  MoveL 1393 to (55.08, -253.68, 406.18) mm, rotated rx -19.35 ry -2.23 rz 0.78 deg; joints [0.707, -147.772, -38.266, -73.505, 93.206, -4.557]
  MoveL 1394 to (54.92, -244.83, 403.1) mm, rotated rx -20.06 ry -2.27 rz 0.83 deg; joints [0.671, -146.589, -40.525, -73.146, 93.202, -4.603]
  MoveL 1395 to (54.92, -237.94, 400.5) mm, rotated rx -20.57 ry -2.12 rz 0.8 deg; joints [0.697, -145.611, -42.376, -72.771, 93.012, -4.583]
  MoveL 1396 to (55.12, -232.38, 398.15) mm, rotated rx -20.87 ry -1.81 rz 0.69 deg; joints [0.778, -144.686, -44.129, -72.215, 92.65, -4.505]
  MoveL 1397 to (55.02, -224.7, 395.11) mm, rotated rx -21.78 ry -1 rz 0.4 deg; joints [1.084, -143.801, -45.655, -72.409, 91.674, -4.211]
  MoveL 1398 to (54.73, -214.72, 391.64) mm, rotated rx -21.72 ry -0.41 rz 0.16 deg; joints [1.286, -141.85, -49.637, -70.273, 91.013, -4.009]
  MoveL 1399 to (54.98, -204.84, 387.37) mm, rotated rx -21.69 ry -0.21 rz 0.08 deg; joints [1.294, -140.064, -53.161, -68.489, 90.801, -4]
  MoveL 1400 to (55.25, -194.58, 383.53) mm, rotated rx -21.83 ry -0.78 rz 0.31 deg; joints [0.986, -138.634, -56.017, -67.249, 91.452, -4.307]
  MoveL 1401 to (55.06, -187.74, 380.29) mm, rotated rx -21.75 ry -1.59 rz 0.63 deg; joints [0.622, -137.594, -58.047, -66.253, 92.371, -4.669]
  MoveL 1402 to (55.53, -182.53, 378.45) mm, rotated rx -21.65 ry -2.04 rz 0.81 deg; joints [0.364, -136.863, -59.574, -65.405, 92.9, -4.926]
  MoveL 1403 to (54.81, -174.44, 375.91) mm, rotated rx -21.54 ry -2.47 rz 0.97 deg; joints [0.18, -135.733, -61.956, -64.088, 93.395, -5.109]
  MoveL 1404 to (54.79, -165.46, 371.7) mm, rotated rx -21.28 ry -2.57 rz 1 deg; joints [0.063, -134.251, -64.859, -62.426, 93.54, -5.222]
  MoveL 1405 to (53.02, -160.4, 369) mm, rotated rx -21.41 ry -2.72 rz 1.07 deg; joints [0.097, -133.514, -66.171, -61.987, 93.684, -5.191]
  MoveL 1406 to (55.23, -155.08, 367) mm, rotated rx -21.73 ry -2.58 rz 1.03 deg; joints [-0.042, -133.026, -67.064, -61.898, 93.535, -5.332]
  MoveL 1407 to (54.71, -145.1, 363.45) mm, rotated rx -21.68 ry -2.38 rz 0.94 deg; joints [0.011, -131.654, -69.821, -60.441, 93.311, -5.278]
  MoveL 1408 to (55.13, -137.69, 360.48) mm, rotated rx -21.26 ry -2.44 rz 0.95 deg; joints [-0.118, -130.495, -72.206, -58.809, 93.424, -5.4]
  MoveL 1409 to (55.28, -132.81, 358.42) mm, rotated rx -20.93 ry -2.36 rz 0.9 deg; joints [-0.148, -129.693, -73.844, -57.645, 93.378, -5.425]
  MoveL 1410 to (55.22, -124.84, 355.82) mm, rotated rx -20.86 ry -2.05 rz 0.78 deg; joints [-0.064, -128.673, -75.93, -56.476, 93.029, -5.339]
  MoveL 1411 to (54.98, -114.49, 352.02) mm, rotated rx -20.31 ry -1.65 rz 0.61 deg; joints [0.034, -127.128, -79.135, -54.23, 92.636, -5.231]
  MoveL 1412 to (59.43, -108.23, 350) mm, rotated rx -20.42 ry -1.45 rz 0.54 deg; joints [-0.284, -126.59, -80.24, -53.769, 92.469, -5.547]
  MoveL 1413 to (54.78, -104.7, 347.81) mm, rotated rx -20.44 ry -1.33 rz 0.49 deg; joints [0.126, -125.933, -81.347, -53.307, 92.267, -5.142]
  MoveL 1414 to (54.83, -96.04, 345.13) mm, rotated rx -20.42 ry -1.17 rz 0.44 deg; joints [0.128, -124.985, -83.305, -52.268, 92.1, -5.139]
  MoveL 1415 to (55.03, -86.29, 340.97) mm, rotated rx -20.38 ry -1.02 rz 0.38 deg; joints [0.101, -123.809, -85.531, -51.167, 91.946, -5.164]
  MoveL 1416 to (55.31, -80.99, 339) mm, rotated rx -20.5 ry -1.09 rz 0.41 deg; joints [0.003, -123.296, -86.506, -50.831, 92.03, -5.263]
  MoveL 1417 to (54.95, -74.37, 337.02) mm, rotated rx -20.6 ry -1.3 rz 0.49 deg; joints [-0.12, -122.697, -87.74, -50.318, 92.266, -5.387]
  MoveL 1418 to (55.01, -64.82, 333.24) mm, rotated rx -20.62 ry -1.46 rz 0.55 deg; joints [-0.287, -121.687, -89.671, -49.444, 92.457, -5.553]
  MoveL 1419 to (54.85, -58, 330.46) mm, rotated rx -20.53 ry -1.63 rz 0.61 deg; joints [-0.429, -120.927, -91.145, -48.659, 92.676, -5.693]
  MoveL 1420 to (55.08, -53.48, 328.66) mm, rotated rx -20.28 ry -1.75 rz 0.65 deg; joints [-0.563, -120.374, -92.289, -47.834, 92.845, -5.822]
  MoveL 1421 to (54.97, -45.34, 325.78) mm, rotated rx -19.8 ry -1.75 rz 0.63 deg; joints [-0.651, -119.376, -94.415, -46.232, 92.899, -5.9]
  MoveL 1422 to (55, -34.77, 321.83) mm, rotated rx -19.25 ry -1.73 rz 0.6 deg; joints [-0.776, -118.117, -97.048, -44.316, 92.948, -6.012]
  MoveL 1423 to (55.17, -28.7, 320) mm, rotated rx -19.04 ry -1.82 rz 0.63 deg; joints [-0.917, -117.517, -98.38, -43.388, 93.099, -6.147]
  MoveL 1424 to (54.83, -23.54, 318) mm, rotated rx -19.21 ry -1.88 rz 0.65 deg; joints [-0.959, -117.05, -99.206, -43.208, 93.144, -6.193]
  MoveL 1425 to (55.14, -14.22, 315.38) mm, rotated rx -19.3 ry -1.62 rz 0.57 deg; joints [-0.947, -116.239, -100.898, -42.396, 92.866, -6.182]
  MoveL 1426 to (54.99, -4.33, 311.44) mm, rotated rx -19.09 ry -1.52 rz 0.53 deg; joints [-1, -115.16, -103.001, -41.15, 92.788, -6.229]
  MoveL 1427 to (55.02, 5.42, 307.78) mm, rotated rx -18.68 ry -1.44 rz 0.49 deg; joints [-1.098, -114.093, -105.207, -39.596, 92.77, -6.316]
  MoveL 1428 to (55.05, 14.94, 305) mm, rotated rx -18.73 ry -1.36 rz 0.46 deg; joints [-1.159, -113.294, -106.879, -38.769, 92.685, -6.377]
  MoveL 1429 to (54.97, 24.93, 302.19) mm, rotated rx -18.4 ry -1.17 rz 0.39 deg; joints [-1.181, -112.36, -108.994, -37.237, 92.527, -6.39]
  MoveL 1430 to (55.25, 31.9, 300) mm, rotated rx -18.6 ry -1.02 rz 0.34 deg; joints [-1.192, -111.805, -110.057, -36.92, 92.345, -6.405]
  MoveL 1431 to (54.96, 36.41, 298.4) mm, rotated rx -18.88 ry -0.94 rz 0.32 deg; joints [-1.157, -111.448, -110.635, -36.964, 92.23, -6.376]
  MoveL 1432 to (54.92, 44.41, 294.89) mm, rotated rx -18.74 ry -0.71 rz 0.24 deg; joints [-1.131, -110.564, -112.252, -36.062, 92.003, -6.347]
  MoveL 1433 to (55.12, 54.76, 291.8) mm, rotated rx -18.4 ry -0.72 rz 0.24 deg; joints [-1.309, -109.656, -114.303, -34.594, 92.079, -6.513]
  MoveL 1434 to (55.11, 61.12, 290) mm, rotated rx -17.74 ry -0.7 rz 0.22 deg; joints [-1.422, -109.017, -115.958, -32.921, 92.152, -6.608]
  MoveL 1435 to (54.8, 66.06, 288.46) mm, rotated rx -17.44 ry -0.7 rz 0.22 deg; joints [-1.477, -108.55, -117.066, -31.98, 92.204, -6.655]
  MoveL 1436 to (54.9, 74.97, 284.68) mm, rotated rx -17.22 ry -0.7 rz 0.22 deg; joints [-1.639, -107.658, -118.76, -30.971, 92.264, -6.807]
  MoveL 1437 to (55.21, 85.34, 282.5) mm, rotated rx -17.34 ry -0.69 rz 0.21 deg; joints [-1.8, -107.029, -120.321, -30.158, 92.267, -6.968]
  MoveL 1438 to (54.78, 93.08, 280.4) mm, rotated rx -17.02 ry -0.27 rz 0.08 deg; joints [-1.61, -106.334, -121.989, -28.813, 91.826, -6.771]
  MoveL 1439 to (57.07, 97.19, 278.81) mm, rotated rx -16.4 ry 0.04 rz -0.01 deg; joints [-1.792, -105.907, -123.158, -27.418, 91.62, -6.931]
  MoveL 1440 to (58.78, 100.67, 277.75) mm, rotated rx -16.4 ry 0.12 rz -0.04 deg; joints [-2.002, -105.698, -123.644, -27.142, 91.586, -7.135]
  MoveL 1441 to (64.56, -260.81, 408.44) mm, rotated rx -18.59 ry -2.72 rz 0.92 deg; joints [-0.095, -149.152, -35.66, -74.064, 93.927, -5.336]
  MoveL 1442 to (65.01, -254.78, 407.2) mm, rotated rx -18.39 ry -2.66 rz 0.88 deg; joints [-0.144, -147.728, -38.763, -72.186, 93.883, -5.38]
  MoveL 1443 to (64.96, -244.73, 403.18) mm, rotated rx -20.08 ry -2.38 rz 0.87 deg; joints [-0.057, -147.081, -39.585, -73.668, 93.443, -5.322]
  MoveL 1444 to (65.61, -236.7, 401.03) mm, rotated rx -21.08 ry -2.09 rz 0.8 deg; joints [-0.012, -146.4, -40.839, -74.057, 93.047, -5.29]
  MoveL 1445 to (62.2, -232.13, 398.8) mm, rotated rx -21.47 ry -1.65 rz 0.65 deg; joints [0.37, -145.511, -42.445, -73.672, 92.498, -4.916]
  MoveL 1446 to (64.8, -224.8, 395.47) mm, rotated rx -22.46 ry -1.21 rz 0.5 deg; joints [0.345, -144.896, -43.381, -74.313, 91.947, -4.951]
  MoveL 1447 to (65.02, -216.02, 391.48) mm, rotated rx -22.19 ry -1.01 rz 0.41 deg; joints [0.343, -142.892, -47.393, -72.019, 91.755, -4.949]
  MoveL 1448 to (67.07, -211.79, 389) mm, rotated rx -22.21 ry -1.04 rz 0.42 deg; joints [0.156, -142.13, -48.809, -71.388, 91.813, -5.134]
  MoveL 1449 to (64.92, -205.17, 386.05) mm, rotated rx -21.61 ry -0.79 rz 0.31 deg; joints [0.347, -140.361, -52.43, -68.915, 91.563, -4.938]
  MoveL 1450 to (64.99, -195.38, 382.72) mm, rotated rx -20.75 ry -1.55 rz 0.59 deg; joints [-0.061, -138.394, -56.676, -65.857, 92.509, -5.332]
  MoveL 1451 to (64.36, -188.78, 380.15) mm, rotated rx -20.94 ry -2.09 rz 0.8 deg; joints [-0.279, -137.586, -58.253, -65.334, 93.099, -5.553]
  MoveL 1452 to (65.35, -183.29, 378.42) mm, rotated rx -21.31 ry -2.24 rz 0.87 deg; joints [-0.445, -137.108, -59.179, -65.283, 93.259, -5.723]
  MoveL 1453 to (65.07, -174.7, 376.9) mm, rotated rx -21.54 ry -2.09 rz 0.83 deg; joints [-0.417, -136.146, -61.303, -64.327, 93.079, -5.698]
  MoveL 1454 to (65.38, -165.59, 372.14) mm, rotated rx -21.23 ry -1.93 rz 0.75 deg; joints [-0.455, -134.518, -64.428, -62.516, 92.93, -5.731]
  MoveL 1455 to (65.07, -160.4, 369) mm, rotated rx -21.45 ry -1.96 rz 0.77 deg; joints [-0.488, -133.793, -65.634, -62.25, 92.959, -5.766]
  MoveL 1456 to (64.92, -155.17, 367.35) mm, rotated rx -21.91 ry -1.93 rz 0.78 deg; joints [-0.486, -133.373, -66.4, -62.362, 92.88, -5.771]
  MoveL 1457 to (65.21, -145.15, 364.29) mm, rotated rx -21.56 ry -2.01 rz 0.79 deg; joints [-0.634, -131.962, -69.413, -60.425, 93.014, -5.914]
  MoveL 1458 to (65.04, -137.22, 360.8) mm, rotated rx -21.12 ry -2.22 rz 0.86 deg; joints [-0.801, -130.701, -71.962, -58.731, 93.304, -6.073]
  MoveL 1459 to (64.64, -132.44, 358.36) mm, rotated rx -21.09 ry -2.27 rz 0.88 deg; joints [-0.84, -130.015, -73.227, -58.128, 93.37, -6.112]
  MoveL 1460 to (65.05, -125.09, 356.02) mm, rotated rx -21.31 ry -2.11 rz 0.82 deg; joints [-0.856, -129.253, -74.741, -57.58, 93.181, -6.13]
  MoveL 1461 to (65.01, -114.69, 352.96) mm, rotated rx -20.63 ry -1.66 rz 0.62 deg; joints [-0.764, -127.702, -78.121, -55.022, 92.744, -6.025]
  MoveL 1462 to (65.64, -107.48, 350.37) mm, rotated rx -20.58 ry -1.42 rz 0.53 deg; joints [-0.776, -126.837, -79.857, -54.086, 92.504, -6.036]
  MoveL 1463 to (65.06, -102.58, 347.84) mm, rotated rx -20.65 ry -1.33 rz 0.5 deg; joints [-0.732, -126.192, -80.984, -53.659, 92.393, -5.992]
  MoveL 1464 to (64.8, -95.29, 344.81) mm, rotated rx -20.52 ry -1.19 rz 0.45 deg; joints [-0.719, -125.245, -82.829, -52.616, 92.255, -5.977]
  MoveL 1465 to (65.28, -85.57, 341) mm, rotated rx -20.49 ry -0.96 rz 0.36 deg; joints [-0.744, -124.11, -85.034, -51.495, 92.02, -6]
  MoveL 1466 to (64.1, -80.02, 339) mm, rotated rx -20.41 ry -0.96 rz 0.36 deg; joints [-0.699, -123.442, -86.371, -50.745, 92.019, -5.955]
  MoveL 1467 to (64.98, -74.27, 337.4) mm, rotated rx -20.3 ry -0.9 rz 0.33 deg; joints [-0.802, -122.854, -87.664, -49.919, 91.98, -6.053]
  MoveL 1468 to (65.02, -64.62, 333.14) mm, rotated rx -20.29 ry -1.17 rz 0.43 deg; joints [-1.039, -121.794, -89.629, -49.048, 92.308, -6.289]
  MoveL 1469 to (65.63, -57.19, 330.53) mm, rotated rx -20.07 ry -1.48 rz 0.54 deg; joints [-1.332, -121.022, -91.254, -48.024, 92.701, -6.575]
  MoveL 1470 to (64.51, -52.14, 329) mm, rotated rx -20.17 ry -1.71 rz 0.63 deg; joints [-1.398, -120.58, -92.152, -47.693, 92.95, -6.644]
  MoveL 1471 to (64.89, -44.96, 327.12) mm, rotated rx -19.87 ry -1.72 rz 0.62 deg; joints [-1.528, -119.845, -93.836, -46.456, 93.013, -6.766]
  MoveL 1472 to (64.91, -34.85, 322.66) mm, rotated rx -19.27 ry -1.62 rz 0.57 deg; joints [-1.632, -118.522, -96.488, -44.523, 92.99, -6.855]
  MoveL 1473 to (65.83, -28.11, 320) mm, rotated rx -19.11 ry -1.5 rz 0.52 deg; joints [-1.744, -117.792, -97.937, -43.641, 92.9, -6.961]
  MoveL 1474 to (64.59, -23.19, 318.3) mm, rotated rx -19.34 ry -1.45 rz 0.51 deg; joints [-1.652, -117.347, -98.733, -43.502, 92.812, -6.875]
  MoveL 1475 to (65.09, -14.35, 315.73) mm, rotated rx -19.48 ry -1.32 rz 0.47 deg; joints [-1.724, -116.61, -100.249, -42.856, 92.668, -6.949]
  MoveL 1476 to (65, -4.36, 312.96) mm, rotated rx -19.17 ry -1.29 rz 0.45 deg; joints [-1.838, -115.661, -102.395, -41.349, 92.691, -7.053]
  MoveL 1477 to (67.12, 1.57, 310) mm, rotated rx -18.88 ry -1.26 rz 0.43 deg; joints [-2.128, -114.98, -103.691, -40.453, 92.745, -7.332]
  MoveL 1478 to (64.74, 5.9, 307.87) mm, rotated rx -18.76 ry -1.19 rz 0.4 deg; joints [-1.922, -114.379, -104.765, -39.846, 92.647, -7.127]
  MoveL 1479 to (64.99, 14.9, 305.22) mm, rotated rx -18.7 ry -1.07 rz 0.36 deg; joints [-2.006, -113.595, -106.445, -38.879, 92.553, -7.206]
  MoveL 1480 to (64.96, 25.12, 302.15) mm, rotated rx -18.59 ry -1.1 rz 0.37 deg; joints [-2.163, -112.716, -108.34, -37.765, 92.624, -7.358]
  MoveL 1481 to (64.3, 31.36, 300) mm, rotated rx -18.81 ry -1.09 rz 0.37 deg; joints [-2.163, -112.197, -109.276, -37.566, 92.587, -7.363]
  MoveL 1482 to (65.2, 36.26, 297.42) mm, rotated rx -19.08 ry -1.06 rz 0.37 deg; joints [-2.298, -111.741, -109.881, -37.689, 92.549, -7.502]
  MoveL 1483 to (65.02, 45.12, 295.08) mm, rotated rx -18.74 ry -1.03 rz 0.35 deg; joints [-2.407, -110.963, -111.72, -36.29, 92.574, -7.602]
  MoveL 1484 to (64.94, 54.73, 292.15) mm, rotated rx -18.47 ry -1.1 rz 0.37 deg; joints [-2.61, -110.134, -113.576, -35.015, 92.73, -7.795]
  MoveL 1485 to (63.94, 60.82, 290) mm, rotated rx -17.96 ry -1.03 rz 0.33 deg; joints [-2.59, -109.442, -115.145, -33.614, 92.712, -7.76]
  MoveL 1486 to (65.16, 65.51, 288.44) mm, rotated rx -17.52 ry -0.96 rz 0.3 deg; joints [-2.795, -108.996, -116.265, -32.505, 92.744, -7.948]
  MoveL 1487 to (64.96, 75.06, 285.39) mm, rotated rx -17.35 ry -0.63 rz 0.2 deg; joints [-2.738, -108.132, -118.107, -31.313, 92.412, -7.884]
  MoveL 1488 to (65.01, 85.34, 282.44) mm, rotated rx -17.3 ry -0.39 rz 0.12 deg; joints [-2.761, -107.319, -119.899, -30.253, 92.171, -7.904]
  MoveL 1489 to (64.71, 92.06, 280.15) mm, rotated rx -17.29 ry -0.5 rz 0.16 deg; joints [-2.917, -106.779, -120.993, -29.708, 92.321, -8.057]
  MoveL 1490 to (65.23, 97.05, 278.32) mm, rotated rx -16.92 ry -0.44 rz 0.13 deg; joints [-3.067, -106.307, -122.11, -28.689, 92.347, -8.191]
  MoveL 1491 to (65.21, 101.45, 276.39) mm, rotated rx -16.78 ry -0.11 rz 0.03 deg; joints [-2.937, -105.802, -123.062, -28.05, 91.99, -8.058]
  MoveL 1492 to (75.11, -263.32, 410.7) mm, rotated rx -19.34 ry -1.95 rz 0.68 deg; joints [-0.467, -151.14, -31.599, -76.835, 93.119, -5.711]
  MoveL 1493 to (80.87, -259.66, 410) mm, rotated rx -18.89 ry -2.65 rz 0.91 deg; joints [-1.154, -150.329, -33.526, -75.386, 94.028, -6.384]
  MoveL 1494 to (75.51, -259.66, 410) mm, rotated rx -18.52 ry -2.32 rz 0.78 deg; joints [-0.683, -149.52, -35.241, -74.043, 93.622, -5.91]
  MoveL 1495 to (75.18, -253.52, 407.14) mm, rotated rx -18.5 ry -2.65 rz 0.89 deg; joints [-0.833, -148.106, -38.068, -72.657, 93.999, -6.06]
  MoveL 1496 to (74.85, -244.56, 402.65) mm, rotated rx -20.82 ry -2.61 rz 0.99 deg; joints [-0.798, -148.266, -36.982, -75.881, 93.751, -6.068]
  MoveL 1497 to (75.1, -236.23, 401.3) mm, rotated rx -21.65 ry -2.25 rz 0.89 deg; joints [-0.706, -147.409, -38.764, -75.751, 93.279, -5.988]
  MoveL 1498 to (75.24, -225.13, 395.22) mm, rotated rx -22.62 ry -2.19 rz 0.91 deg; joints [-0.755, -145.769, -41.608, -75.508, 93.139, -6.049]
  MoveL 1499 to (75.24, -216.09, 391.13) mm, rotated rx -22.66 ry -1.94 rz 0.81 deg; joints [-0.725, -143.894, -45.288, -73.718, 92.856, -6.018]
  MoveL 1500 to (73.17, -211.79, 389) mm, rotated rx -22.42 ry -1.54 rz 0.64 deg; joints [-0.465, -142.659, -47.738, -72.212, 92.417, -5.755]
  MoveL 1501 to (75.03, -204.96, 386.98) mm, rotated rx -21.4 ry -1.74 rz 0.68 deg; joints [-0.76, -140.874, -51.676, -69.076, 92.76, -6.034]
  MoveL 1502 to (75.1, -194.69, 383.85) mm, rotated rx -20.24 ry -1.83 rz 0.67 deg; joints [-0.922, -138.535, -56.799, -65.146, 92.989, -6.176]
  MoveL 1503 to (75.37, -187.45, 380.54) mm, rotated rx -20.91 ry -1.7 rz 0.65 deg; joints [-0.928, -137.788, -58.037, -65.311, 92.79, -6.192]
  MoveL 1504 to (74.68, -182.22, 378.28) mm, rotated rx -21.5 ry -1.62 rz 0.64 deg; joints [-0.87, -137.312, -58.79, -65.613, 92.643, -6.144]
  MoveL 1505 to (74.95, -174.56, 376.81) mm, rotated rx -21.88 ry -1.3 rz 0.52 deg; joints [-0.797, -136.526, -60.478, -65.05, 92.246, -6.076]
  MoveL 1506 to (75.03, -164.4, 371.69) mm, rotated rx -21.14 ry -0.97 rz 0.37 deg; joints [-0.783, -134.451, -64.613, -62.222, 91.966, -6.049]
  MoveL 1507 to (75.88, -158.9, 370) mm, rotated rx -21.36 ry -0.93 rz 0.36 deg; joints [-0.869, -133.892, -65.735, -61.876, 91.919, -6.138]
  MoveL 1508 to (74.82, -154.25, 367.84) mm, rotated rx -21.66 ry -1.25 rz 0.5 deg; joints [-0.956, -133.412, -66.553, -61.873, 92.243, -6.23]
  MoveL 1509 to (75.16, -145.64, 365.57) mm, rotated rx -21.37 ry -1.63 rz 0.64 deg; joints [-1.23, -132.313, -68.983, -60.309, 92.714, -6.499]
  MoveL 1510 to (75.18, -136.04, 361.41) mm, rotated rx -21.02 ry -1.56 rz 0.6 deg; joints [-1.311, -130.841, -71.918, -58.497, 92.692, -6.572]
  MoveL 1511 to (74.07, -131.61, 358.88) mm, rotated rx -21.06 ry -1.58 rz 0.61 deg; joints [-1.277, -130.175, -73.085, -58.029, 92.702, -6.54]
  MoveL 1512 to (74.88, -125, 356.05) mm, rotated rx -21.49 ry -1.58 rz 0.62 deg; joints [-1.388, -129.57, -74.116, -58.043, 92.675, -6.657]
  MoveL 1513 to (75.04, -114.51, 352.44) mm, rotated rx -21.12 ry -1.33 rz 0.51 deg; joints [-1.405, -128.125, -77.123, -56.081, 92.447, -6.666]
  MoveL 1514 to (74.03, -107.97, 350.43) mm, rotated rx -20.83 ry -1.07 rz 0.41 deg; joints [-1.282, -127.196, -79.103, -54.703, 92.187, -6.538]
  MoveL 1515 to (75.51, -103.23, 347.77) mm, rotated rx -20.74 ry -0.91 rz 0.35 deg; joints [-1.385, -126.535, -80.291, -54.079, 92.043, -6.638]
  MoveL 1516 to (75, -94.89, 345.05) mm, rotated rx -20.65 ry -0.85 rz 0.32 deg; joints [-1.402, -125.565, -82.294, -52.943, 91.988, -6.652]
  MoveL 1517 to (74.92, -84.51, 341.34) mm, rotated rx -20.72 ry -0.72 rz 0.27 deg; joints [-1.437, -124.438, -84.516, -51.909, 91.848, -6.688]
  MoveL 1518 to (75.1, -74.48, 337.81) mm, rotated rx -20.46 ry -0.55 rz 0.21 deg; joints [-1.49, -123.242, -86.983, -50.358, 91.706, -6.735]
  MoveL 1519 to (75, -64.84, 333.79) mm, rotated rx -19.97 ry -0.47 rz 0.17 deg; joints [-1.578, -121.963, -89.57, -48.554, 91.696, -6.811]
  MoveL 1520 to (75.02, -56.43, 330.96) mm, rotated rx -19.78 ry -0.67 rz 0.24 deg; joints [-1.78, -121.084, -91.416, -47.426, 91.958, -7.007]
  MoveL 1521 to (74.42, -51.73, 329) mm, rotated rx -19.89 ry -0.86 rz 0.31 deg; joints [-1.874, -120.632, -92.222, -47.219, 92.165, -7.103]
  MoveL 1522 to (75.01, -45.45, 326.52) mm, rotated rx -19.84 ry -0.94 rz 0.34 deg; joints [-2.045, -119.987, -93.482, -46.568, 92.283, -7.27]
  MoveL 1523 to (75.01, -34.99, 324.07) mm, rotated rx -19.45 ry -0.83 rz 0.29 deg; joints [-2.135, -118.954, -95.906, -44.775, 92.234, -7.35]
  MoveL 1524 to (74.93, -27.07, 320.43) mm, rotated rx -19.19 ry -0.7 rz 0.24 deg; joints [-2.178, -117.977, -97.768, -43.622, 92.129, -7.385]
  MoveL 1525 to (74.92, -21.92, 318.61) mm, rotated rx -19.29 ry -0.81 rz 0.28 deg; joints [-2.299, -117.533, -98.621, -43.325, 92.261, -7.507]
  MoveL 1526 to (75.04, -14.29, 315.6) mm, rotated rx -19.5 ry -0.98 rz 0.35 deg; joints [-2.488, -116.867, -99.812, -43.038, 92.444, -7.7]
  MoveL 1527 to (74.96, -4.46, 312.76) mm, rotated rx -19.02 ry -1.05 rz 0.36 deg; joints [-2.685, -115.891, -102.049, -41.327, 92.621, -7.882]
  MoveL 1528 to (75.69, 3.3, 310) mm, rotated rx -19.07 ry -0.99 rz 0.34 deg; joints [-2.829, -115.198, -103.408, -40.705, 92.572, -8.024]
  MoveL 1529 to (74.23, 7.81, 308.64) mm, rotated rx -18.97 ry -0.95 rz 0.33 deg; joints [-2.736, -114.727, -104.41, -40.063, 92.529, -7.93]
  MoveL 1530 to (74.94, 14.96, 305.92) mm, rotated rx -18.83 ry -0.86 rz 0.29 deg; joints [-2.875, -114.021, -105.828, -39.204, 92.482, -8.062]
  MoveL 1531 to (74.99, 25.08, 302.55) mm, rotated rx -18.4 ry -0.92 rz 0.31 deg; joints [-3.101, -113.04, -107.984, -37.628, 92.647, -8.273]
  MoveL 1532 to (76.15, 31.98, 300.05) mm, rotated rx -18.82 ry -1.04 rz 0.36 deg; joints [-3.368, -112.587, -108.722, -37.782, 92.764, -8.547]
  MoveL 1533 to (74.3, 36.05, 298.14) mm, rotated rx -19.01 ry -1.09 rz 0.37 deg; joints [-3.257, -112.153, -109.372, -37.758, 92.761, -8.444]
  MoveL 1534 to (75.11, 44.67, 295.69) mm, rotated rx -18.62 ry -1.21 rz 0.41 deg; joints [-3.586, -111.431, -111.107, -36.397, 93.009, -8.758]
  MoveL 1535 to (74.88, 54.68, 291.77) mm, rotated rx -18.37 ry -1.5 rz 0.5 deg; joints [-3.935, -110.497, -112.979, -35.272, 93.415, -9.096]
  MoveL 1536 to (74.13, 60.4, 290) mm, rotated rx -18.17 ry -1.49 rz 0.49 deg; joints [-3.97, -109.967, -114.156, -34.433, 93.443, -9.124]
  MoveL 1537 to (75.11, 64.93, 288.79) mm, rotated rx -18.05 ry -1.28 rz 0.42 deg; joints [-4.04, -109.604, -115.028, -33.769, 93.255, -9.186]
  MoveL 1538 to (74.84, 75.3, 285.59) mm, rotated rx -17.67 ry -0.8 rz 0.25 deg; joints [-3.939, -108.617, -117.239, -32.091, 92.792, -9.071]
  MoveL 1539 to (75.02, 85.38, 282.27) mm, rotated rx -17.28 ry -0.74 rz 0.23 deg; joints [-4.16, -107.739, -119.233, -30.587, 92.845, -9.273]
  MoveL 1540 to (75.39, 92.51, 280.32) mm, rotated rx -17.48 ry -0.57 rz 0.18 deg; joints [-4.21, -107.252, -120.243, -30.241, 92.644, -9.328]
  MoveL 1541 to (73.93, 97.03, 278.51) mm, rotated rx -17.35 ry -0.42 rz 0.13 deg; joints [-4.047, -106.74, -121.234, -29.597, 92.474, -9.162]
  MoveL 1542 to (73.9, 100.81, 277.62) mm, rotated rx -17.26 ry -0.3 rz 0.09 deg; joints [-4.05, -106.463, -121.947, -29.052, 92.369, -9.161]
  MoveL 1543 to (84.62, -262.23, 410) mm, rotated rx -19.74 ry -3.1 rz 1.11 deg; joints [-1.525, -152.298, -29.177, -78.689, 94.488, -6.771]
  MoveL 1544 to (85.18, -254.45, 406.95) mm, rotated rx -19.33 ry -3.17 rz 1.11 deg; joints [-1.669, -149.81, -34.361, -75.601, 94.625, -6.905]
  MoveL 1545 to (84.93, -244.07, 403.5) mm, rotated rx -21.32 ry -2.99 rz 1.16 deg; joints [-1.6, -149.493, -34.573, -77.657, 94.224, -6.875]
  MoveL 1546 to (84.92, -235.7, 402.03) mm, rotated rx -22.08 ry -2.73 rz 1.11 deg; joints [-1.539, -148.503, -36.641, -77.308, 93.863, -6.824]
  MoveL 1547 to (84.8, -224.66, 395.97) mm, rotated rx -22.6 ry -2.59 rz 1.08 deg; joints [-1.562, -146.344, -40.642, -75.969, 93.667, -6.854]
  MoveL 1548 to (85.07, -214.39, 391.74) mm, rotated rx -22.83 ry -2.65 rz 1.12 deg; joints [-1.688, -144.494, -44.298, -74.403, 93.726, -6.983]
  MoveL 1549 to (86.97, -207.97, 390) mm, rotated rx -21.77 ry -3 rz 1.2 deg; joints [-2.055, -142.69, -48.316, -71.198, 94.257, -7.334]
  MoveL 1550 to (90.52, -207.58, 390) mm, rotated rx -21.73 ry -3.09 rz 1.23 deg; joints [-2.341, -142.798, -48.151, -71.253, 94.395, -7.619]
  MoveL 1551 to (84.6, -203.52, 388.23) mm, rotated rx -21.16 ry -2.83 rz 1.1 deg; joints [-1.888, -141.306, -51.227, -69.033, 94.118, -7.156]
  MoveL 1552 to (85.05, -194.33, 384.67) mm, rotated rx -20.74 ry -2.35 rz 0.89 deg; joints [-1.83, -139.426, -55.091, -66.575, 93.638, -7.086]
  MoveL 1553 to (85.62, -185.53, 380.69) mm, rotated rx -21.69 ry -1.5 rz 0.6 deg; joints [-1.569, -138.461, -56.672, -66.792, 92.592, -6.84]
  MoveL 1554 to (83.88, -181.16, 378.92) mm, rotated rx -22.09 ry -1.17 rz 0.48 deg; joints [-1.332, -137.911, -57.642, -66.725, 92.163, -6.609]
  MoveL 1555 to (85.03, -174.6, 376.81) mm, rotated rx -22.34 ry -0.68 rz 0.28 deg; joints [-1.258, -137.07, -59.321, -66.066, 91.599, -6.537]
  MoveL 1556 to (85.14, -164.6, 371.9) mm, rotated rx -21.31 ry -0.54 rz 0.21 deg; joints [-1.346, -134.868, -63.812, -62.74, 91.573, -6.607]
  MoveL 1557 to (85.07, -158.9, 370) mm, rotated rx -21.03 ry -0.63 rz 0.24 deg; joints [-1.446, -133.974, -65.713, -61.469, 91.721, -6.701]
  MoveL 1558 to (85.04, -154.1, 367.79) mm, rotated rx -20.99 ry -0.8 rz 0.31 deg; joints [-1.563, -133.299, -67.009, -60.834, 91.917, -6.817]
  MoveL 1559 to (85.13, -145.29, 365.23) mm, rotated rx -21.13 ry -1.21 rz 0.47 deg; joints [-1.827, -132.389, -68.917, -60.035, 92.387, -7.083]
  MoveL 1560 to (84.92, -135.28, 361.14) mm, rotated rx -21.24 ry -1.25 rz 0.48 deg; joints [-1.923, -131.137, -71.329, -58.997, 92.422, -7.181]
  MoveL 1561 to (84.88, -124.93, 356.15) mm, rotated rx -21.55 ry -1 rz 0.4 deg; joints [-1.912, -129.839, -73.641, -58.257, 92.126, -7.174]
  MoveL 1562 to (85, -114.4, 352.4) mm, rotated rx -21.39 ry -0.85 rz 0.33 deg; joints [-1.971, -128.491, -76.384, -56.687, 91.991, -7.229]
  MoveL 1563 to (85.47, -107.67, 350.29) mm, rotated rx -21.16 ry -0.75 rz 0.29 deg; joints [-2.047, -127.64, -78.203, -55.483, 91.924, -7.299]
  MoveL 1564 to (84.68, -102.56, 348.03) mm, rotated rx -21.01 ry -0.59 rz 0.23 deg; joints [-1.973, -126.884, -79.671, -54.597, 91.757, -7.223]
  MoveL 1565 to (84.73, -94.7, 345.08) mm, rotated rx -20.69 ry -0.4 rz 0.15 deg; joints [-1.994, -125.818, -81.869, -53.117, 91.598, -7.236]
  MoveL 1566 to (85.2, -84.82, 341.13) mm, rotated rx -20.7 ry -0.44 rz 0.17 deg; joints [-2.164, -124.718, -83.994, -52.114, 91.664, -7.404]
  MoveL 1567 to (85.17, -74.33, 337.43) mm, rotated rx -20.66 ry -0.5 rz 0.19 deg; joints [-2.315, -123.596, -86.253, -50.952, 91.758, -7.553]
  MoveL 1568 to (84.97, -64.89, 333.9) mm, rotated rx -20.2 ry -0.07 rz 0.03 deg; joints [-2.233, -122.329, -88.878, -49.076, 91.354, -7.46]
  MoveL 1569 to (84.98, -56.59, 331.06) mm, rotated rx -19.62 ry 0.22 rz -0.08 deg; joints [-2.226, -121.234, -91.26, -47.177, 91.122, -7.44]
  MoveL 1570 to (85.06, -51.84, 328.83) mm, rotated rx -19.58 ry 0.11 rz -0.04 deg; joints [-2.351, -120.695, -92.251, -46.695, 91.262, -7.561]
  MoveL 1571 to (85.07, -45.47, 326.64) mm, rotated rx -19.64 ry -0.11 rz 0.04 deg; joints [-2.538, -120.128, -93.373, -46.24, 91.516, -7.748]
  MoveL 1572 to (85.07, -35, 324) mm, rotated rx -19.61 ry -0.34 rz 0.12 deg; joints [-2.79, -119.257, -95.33, -45.167, 91.809, -7.997]
  MoveL 1573 to (84.43, -27.54, 320.55) mm, rotated rx -19.07 ry -0.49 rz 0.17 deg; joints [-2.954, -118.266, -97.328, -43.649, 92.071, -8.144]
  MoveL 1574 to (85.15, -22.51, 318.39) mm, rotated rx -19.02 ry -0.56 rz 0.19 deg; joints [-3.138, -117.763, -98.28, -43.174, 92.191, -8.325]
  MoveL 1575 to (85.09, -14.25, 315.9) mm, rotated rx -19.33 ry -0.59 rz 0.21 deg; joints [-3.244, -117.132, -99.515, -42.88, 92.198, -8.437]
  MoveL 1576 to (84.98, -4.26, 312.2) mm, rotated rx -18.98 ry -0.91 rz 0.31 deg; joints [-3.583, -116.127, -101.611, -41.509, 92.644, -8.763]
  MoveL 1577 to (82.62, 2.29, 310) mm, rotated rx -19.05 ry -1.02 rz 0.35 deg; joints [-3.512, -115.492, -102.844, -40.993, 92.738, -8.696]
  MoveL 1578 to (85.48, 6.19, 308.36) mm, rotated rx -19.06 ry -1.13 rz 0.39 deg; joints [-3.912, -115.227, -103.352, -40.796, 92.92, -9.091]
  MoveL 1579 to (84.99, 14.95, 306.4) mm, rotated rx -18.9 ry -1.12 rz 0.38 deg; joints [-4.009, -114.512, -105.069, -39.637, 92.952, -9.182]
  MoveL 1580 to (84.93, 24.98, 302.2) mm, rotated rx -18.3 ry -1.09 rz 0.36 deg; joints [-4.217, -113.368, -107.434, -37.833, 93.055, -9.367]
  MoveL 1581 to (84.61, 32.85, 300.05) mm, rotated rx -18.72 ry -1.15 rz 0.39 deg; joints [-4.316, -112.86, -108.411, -37.792, 93.066, -9.478]
  MoveL 1582 to (85.33, 37.25, 298.87) mm, rotated rx -18.93 ry -1.25 rz 0.43 deg; joints [-4.512, -112.623, -108.9, -37.773, 93.184, -9.678]
  MoveL 1583 to (85.08, 44.63, 296.09) mm, rotated rx -18.5 ry -1.28 rz 0.43 deg; joints [-4.681, -111.847, -110.573, -36.465, 93.312, -9.831]
  MoveL 1584 to (85.01, 54.71, 292.37) mm, rotated rx -18.28 ry -1.28 rz 0.42 deg; joints [-4.894, -110.904, -112.497, -35.28, 93.39, -10.032]
  MoveL 1585 to (85.16, 61.25, 290.32) mm, rotated rx -18.54 ry -1.06 rz 0.36 deg; joints [-4.885, -110.403, -113.436, -35.055, 93.12, -10.03]
  MoveL 1586 to (84.98, 66.19, 288.57) mm, rotated rx -18.39 ry -0.9 rz 0.3 deg; joints [-4.88, -109.912, -114.461, -34.349, 92.971, -10.019]
  MoveL 1587 to (84.99, 75.45, 285.6) mm, rotated rx -17.77 ry -0.97 rz 0.31 deg; joints [-5.182, -109.067, -116.499, -32.569, 93.218, -10.294]
  MoveL 1588 to (85.09, 85.49, 282.27) mm, rotated rx -17.69 ry -0.89 rz 0.29 deg; joints [-5.37, -108.242, -118.228, -31.586, 93.187, -10.474]
  MoveL 1589 to (85, 93.4, 280.15) mm, rotated rx -17.7 ry -0.79 rz 0.25 deg; joints [-5.468, -107.671, -119.528, -30.849, 93.103, -10.569]
  MoveL 1590 to (84.49, 97.29, 279) mm, rotated rx -17.6 ry -0.77 rz 0.24 deg; joints [-5.489, -107.347, -120.271, -30.332, 93.095, -10.585]
  MoveL 1591 to (93.64, -252.15, 406.29) mm, rotated rx -19.83 ry -3.26 rz 1.18 deg; joints [-2.269, -150.38, -33.145, -76.804, 94.776, -7.511]
  MoveL 1592 to (94.89, -244.5, 404.61) mm, rotated rx -21.46 ry -3.07 rz 1.21 deg; joints [-2.283, -150.53, -32.607, -78.79, 94.394, -7.556]
  MoveL 1593 to (94.98, -234.81, 402.26) mm, rotated rx -22.55 ry -2.8 rz 1.16 deg; joints [-2.229, -149.478, -34.684, -78.805, 93.981, -7.519]
  MoveL 1594 to (95.1, -223.99, 396.31) mm, rotated rx -22.44 ry -2.6 rz 1.07 deg; joints [-2.275, -146.658, -40.179, -75.999, 93.782, -7.561]
  MoveL 1595 to (94.94, -214.19, 391.71) mm, rotated rx -22.53 ry -2.76 rz 1.14 deg; joints [-2.421, -144.714, -43.981, -74.266, 93.96, -7.709]
  MoveL 1596 to (95.36, -204.14, 388.29) mm, rotated rx -21.51 ry -2.74 rz 1.08 deg; joints [-2.587, -142.119, -49.526, -70.313, 94.083, -7.855]
  MoveL 1597 to (95.03, -194.48, 384.9) mm, rotated rx -21.78 ry -2.09 rz 0.83 deg; joints [-2.386, -140.554, -52.634, -68.939, 93.321, -7.655]
  MoveL 1598 to (94.62, -185.05, 380.97) mm, rotated rx -22.51 ry -1.26 rz 0.52 deg; joints [-2.085, -139.309, -54.888, -68.535, 92.313, -7.363]
  MoveL 1599 to (97.05, -180.59, 379) mm, rotated rx -22.65 ry -1.32 rz 0.55 deg; joints [-2.323, -138.793, -55.868, -68.225, 92.393, -7.603]
  MoveL 1600 to (94.6, -174.94, 376.31) mm, rotated rx -22.5 ry -1.22 rz 0.51 deg; joints [-2.172, -137.648, -58.101, -66.97, 92.283, -7.449]
  MoveL 1601 to (95.24, -165.19, 371.54) mm, rotated rx -21.32 ry -1.37 rz 0.53 deg; joints [-2.443, -135.447, -62.642, -63.492, 92.622, -7.697]
  MoveL 1602 to (94.74, -158.9, 370) mm, rotated rx -21.14 ry -1.24 rz 0.48 deg; joints [-2.424, -134.519, -64.67, -62.189, 92.507, -7.675]
  MoveL 1603 to (95.18, -154.18, 367.97) mm, rotated rx -21.13 ry -1.06 rz 0.41 deg; joints [-2.433, -133.831, -66.008, -61.508, 92.316, -7.682]
  MoveL 1604 to (95.01, -145.33, 364.77) mm, rotated rx -20.87 ry -1.05 rz 0.4 deg; joints [-2.523, -132.538, -68.68, -59.877, 92.347, -7.765]
  MoveL 1605 to (94.91, -135.39, 361.45) mm, rotated rx -21.3 ry -1.21 rz 0.47 deg; joints [-2.673, -131.566, -70.574, -59.402, 92.488, -7.924]
  MoveL 1606 to (95.24, -125.63, 357.23) mm, rotated rx -21.71 ry -1.13 rz 0.45 deg; joints [-2.756, -130.492, -72.515, -58.934, 92.361, -8.014]
  MoveL 1607 to (95.03, -114.74, 353.13) mm, rotated rx -21.48 ry -1.09 rz 0.43 deg; joints [-2.864, -129.044, -75.447, -57.222, 92.365, -8.116]
  MoveL 1608 to (94.04, -107.45, 350.45) mm, rotated rx -21.3 ry -0.88 rz 0.34 deg; joints [-2.787, -128.032, -77.497, -55.98, 92.152, -8.034]
  MoveL 1609 to (95.5, -102.51, 348) mm, rotated rx -21.19 ry -0.83 rz 0.32 deg; joints [-2.951, -127.384, -78.722, -55.29, 92.139, -8.195]
  MoveL 1610 to (95.46, -94.69, 345.35) mm, rotated rx -21.08 ry -0.64 rz 0.25 deg; joints [-2.964, -126.436, -80.675, -54.144, 91.955, -8.204]
  MoveL 1611 to (94.7, -85.12, 341.38) mm, rotated rx -20.66 ry -0.32 rz 0.12 deg; joints [-2.9, -125.059, -83.439, -52.289, 91.664, -8.129]
  MoveL 1612 to (95.22, -80.02, 339) mm, rotated rx -20.64 ry -0.25 rz 0.1 deg; joints [-2.981, -124.448, -84.568, -51.751, 91.608, -8.209]
  MoveL 1613 to (95.02, -74.21, 336.71) mm, rotated rx -20.97 ry -0.14 rz 0.06 deg; joints [-2.967, -123.912, -85.503, -51.664, 91.444, -8.202]
  MoveL 1614 to (95.11, -64.87, 333.68) mm, rotated rx -20.61 ry 0.02 rz -0.01 deg; joints [-3.038, -122.794, -87.89, -50.008, 91.331, -8.263]
  MoveL 1615 to (95.03, -56.45, 330.98) mm, rotated rx -19.66 ry 0.12 rz -0.04 deg; joints [-3.158, -121.594, -90.634, -47.514, 91.387, -8.358]
  MoveL 1616 to (94.97, -51.85, 328.91) mm, rotated rx -19.33 ry 0.11 rz -0.04 deg; joints [-3.247, -120.963, -91.92, -46.532, 91.462, -8.436]
  MoveL 1617 to (95.01, -45.5, 326.38) mm, rotated rx -19.23 ry -0.12 rz 0.04 deg; joints [-3.466, -120.309, -93.21, -45.841, 91.76, -8.65]
  MoveL 1618 to (94.86, -34.86, 322.71) mm, rotated rx -19.23 ry -0.73 rz 0.25 deg; joints [-3.917, -119.387, -95.078, -45.015, 92.479, -9.097]
  MoveL 1619 to (95.21, -27.93, 320.36) mm, rotated rx -18.93 ry -1.01 rz 0.35 deg; joints [-4.224, -118.7, -96.59, -43.947, 92.878, -9.393]
  MoveL 1620 to (94.88, -22.66, 318.14) mm, rotated rx -19.15 ry -0.94 rz 0.33 deg; joints [-4.228, -118.201, -97.429, -43.817, 92.771, -9.403]
  MoveL 1621 to (94.97, -14.36, 315.85) mm, rotated rx -19.2 ry -0.85 rz 0.29 deg; joints [-4.314, -117.495, -98.949, -43.036, 92.678, -9.488]
  MoveL 1622 to (95.02, -4.3, 312.79) mm, rotated rx -18.76 ry -1.05 rz 0.36 deg; joints [-4.63, -116.534, -101.133, -41.437, 93.02, -9.787]
  MoveL 1623 to (95.61, 1.36, 310.1) mm, rotated rx -18.79 ry -1.17 rz 0.4 deg; joints [-4.854, -115.983, -102.09, -41.093, 93.181, -10.009]
  MoveL 1624 to (94.88, 6.06, 307.95) mm, rotated rx -19.04 ry -1.21 rz 0.42 deg; joints [-4.872, -115.544, -102.761, -41.114, 93.183, -10.035]
  MoveL 1625 to (94.84, 14.8, 305.86) mm, rotated rx -18.83 ry -1.2 rz 0.41 deg; joints [-5.035, -114.819, -104.495, -39.906, 93.242, -10.189]
  MoveL 1626 to (94.96, 25.02, 302.3) mm, rotated rx -18.41 ry -1.09 rz 0.36 deg; joints [-5.218, -113.788, -106.723, -38.281, 93.233, -10.353]
  MoveL 1627 to (95.09, 32.35, 300.06) mm, rotated rx -18.48 ry -1.07 rz 0.36 deg; joints [-5.354, -113.209, -107.931, -37.721, 93.225, -10.489]
  MoveL 1628 to (95.04, 36.7, 298.67) mm, rotated rx -18.75 ry -1.11 rz 0.38 deg; joints [-5.433, -112.923, -108.423, -37.8, 93.236, -10.577]
  MoveL 1629 to (95.1, 44.75, 296.57) mm, rotated rx -18.65 ry -0.99 rz 0.33 deg; joints [-5.537, -112.279, -109.912, -36.841, 93.149, -10.675]
  MoveL 1630 to (95.08, 54.87, 292.96) mm, rotated rx -18.43 ry -0.72 rz 0.24 deg; joints [-5.615, -111.303, -111.935, -35.524, 92.927, -10.74]
  MoveL 1631 to (95.43, 62.47, 290.4) mm, rotated rx -18.53 ry -0.89 rz 0.3 deg; joints [-5.905, -110.748, -113.037, -35.128, 93.138, -11.031]
  MoveL 1632 to (94.7, 67.27, 288.48) mm, rotated rx -18.16 ry -1.04 rz 0.34 deg; joints [-6.067, -110.236, -114.158, -34.197, 93.396, -11.178]
  MoveL 1633 to (94.76, 74.85, 285.94) mm, rotated rx -17.69 ry -1.07 rz 0.34 deg; joints [-6.317, -109.54, -115.801, -32.8, 93.563, -11.404]
  MoveL 1634 to (95.2, 84.98, 282.66) mm, rotated rx -17.83 ry -0.94 rz 0.3 deg; joints [-6.509, -108.77, -117.353, -32.139, 93.44, -11.596]
  MoveL 1635 to (95.17, 93.09, 280.42) mm, rotated rx -17.81 ry -0.96 rz 0.31 deg; joints [-6.715, -108.203, -118.657, -31.399, 93.505, -11.798]
  MoveL 1636 to (95.06, 97.29, 278.97) mm, rotated rx -17.94 ry -1.01 rz 0.33 deg; joints [-6.823, -107.899, -119.21, -31.301, 93.55, -11.91]
  MoveL 1637 to (98.11, 102.1, 277.5) mm, rotated rx -18.34 ry -1.02 rz 0.34 deg; joints [-7.256, -107.753, -119.434, -31.639, 93.573, -12.352]
  MoveL 1638 to (108.72, -260.92, 412) mm, rotated rx -17.85 ry -3.72 rz 1.2 deg; joints [-3.42, -151.827, -31.148, -75.551, 95.697, -8.601]
  MoveL 1639 to (107.34, -257.32, 410.83) mm, rotated rx -18.67 ry -3.42 rz 1.16 deg; joints [-3.22, -151.672, -31.245, -76.364, 95.243, -8.423]
  MoveL 1640 to (103.45, -252.09, 408.17) mm, rotated rx -19.77 ry -3.17 rz 1.14 deg; joints [-2.88, -151.159, -31.879, -77.267, 94.788, -8.113]
  MoveL 1641 to (104.95, -245.64, 406.26) mm, rotated rx -21.13 ry -2.93 rz 1.13 deg; joints [-2.895, -151.203, -31.527, -78.892, 94.373, -8.155]
  MoveL 1642 to (104.92, -234.64, 402.05) mm, rotated rx -22.87 ry -2.7 rz 1.14 deg; joints [-2.842, -150.388, -32.787, -80.141, 93.908, -8.132]
  MoveL 1643 to (105.01, -224.78, 397.15) mm, rotated rx -22.75 ry -2.17 rz 0.91 deg; joints [-2.755, -147.628, -38.255, -77.24, 93.343, -8.039]
  MoveL 1644 to (104.88, -214.91, 392.63) mm, rotated rx -22.47 ry -1.93 rz 0.8 deg; joints [-2.77, -145.157, -43.215, -74.442, 93.124, -8.048]
  MoveL 1645 to (107.13, -207.7, 390.1) mm, rotated rx -21.86 ry -1.85 rz 0.74 deg; joints [-2.997, -143.403, -46.951, -71.852, 93.148, -8.261]
  MoveL 1646 to (104.25, -203.57, 388.41) mm, rotated rx -21.81 ry -1.89 rz 0.75 deg; joints [-2.857, -142.484, -48.787, -70.88, 93.169, -8.121]
  MoveL 1647 to (105.05, -194.66, 385.2) mm, rotated rx -22.26 ry -1.6 rz 0.65 deg; joints [-2.869, -141.292, -51.113, -70.156, 92.804, -8.14]
  MoveL 1648 to (104.9, -185.62, 381.03) mm, rotated rx -22.66 ry -1.65 rz 0.69 deg; joints [-2.963, -140.025, -53.465, -69.478, 92.824, -8.241]
  MoveL 1649 to (104.83, -180.77, 379) mm, rotated rx -22.45 ry -1.72 rz 0.71 deg; joints [-3.052, -139.11, -55.325, -68.346, 92.937, -8.326]
  MoveL 1650 to (104.78, -175.49, 376.55) mm, rotated rx -22.28 ry -1.87 rz 0.77 deg; joints [-3.181, -138.172, -57.188, -67.282, 93.137, -8.451]
  MoveL 1651 to (104.67, -165.18, 371.25) mm, rotated rx -21.5 ry -1.83 rz 0.72 deg; joints [-3.322, -136.002, -61.518, -64.344, 93.213, -8.575]
  MoveL 1652 to (105.22, -158.57, 370) mm, rotated rx -21.39 ry -1.74 rz 0.68 deg; joints [-3.404, -135.16, -63.427, -63.162, 93.151, -8.654]
  MoveL 1653 to (104.51, -154.03, 367.93) mm, rotated rx -21.28 ry -1.62 rz 0.63 deg; joints [-3.36, -134.383, -64.946, -62.291, 93.022, -8.607]
  MoveL 1654 to (105.06, -145.3, 365.16) mm, rotated rx -20.84 ry -1.52 rz 0.58 deg; joints [-3.486, -133.047, -67.817, -60.31, 92.996, -8.721]
  MoveL 1655 to (104.7, -136.02, 361.44) mm, rotated rx -21.23 ry -1.5 rz 0.58 deg; joints [-3.545, -132.02, -69.725, -59.817, 92.93, -8.788]
  MoveL 1656 to (106, -131.65, 359) mm, rotated rx -21.47 ry -1.53 rz 0.6 deg; joints [-3.706, -131.565, -70.45, -59.8, 92.956, -8.953]
  MoveL 1657 to (105.2, -125.53, 357.26) mm, rotated rx -21.66 ry -1.48 rz 0.59 deg; joints [-3.686, -130.917, -71.778, -59.296, 92.872, -8.937]
  MoveL 1658 to (105.01, -114.82, 353.45) mm, rotated rx -21.84 ry -1.08 rz 0.43 deg; joints [-3.619, -129.634, -74.305, -58.163, 92.404, -8.871]
  MoveL 1659 to (104.71, -108.23, 350) mm, rotated rx -21.58 ry -0.91 rz 0.36 deg; joints [-3.627, -128.571, -76.316, -56.932, 92.263, -8.873]
  MoveL 1660 to (104.86, -103.07, 347.79) mm, rotated rx -21.39 ry -0.79 rz 0.31 deg; joints [-3.67, -127.831, -77.79, -55.989, 92.179, -8.91]
  MoveL 1661 to (105.15, -94.24, 344.95) mm, rotated rx -21.23 ry -0.73 rz 0.28 deg; joints [-3.79, -126.798, -79.959, -54.687, 92.15, -9.025]
  MoveL 1662 to (105.21, -84.58, 341.53) mm, rotated rx -20.97 ry -0.62 rz 0.24 deg; joints [-3.896, -125.611, -82.415, -53.148, 92.093, -9.123]
  MoveL 1663 to (101.86, -80.02, 339) mm, rotated rx -20.86 ry -0.29 rz 0.11 deg; joints [-3.54, -124.785, -83.9, -52.319, 91.704, -8.766]
  MoveL 1664 to (108.39, -78.48, 340) mm, rotated rx -21.04 ry -0.83 rz 0.32 deg; joints [-4.333, -125.218, -83.336, -52.742, 92.366, -9.558]
  MoveL 1665 to (104.76, -74.06, 337.28) mm, rotated rx -21.01 ry -0.4 rz 0.15 deg; joints [-3.905, -124.384, -84.764, -52.033, 91.856, -9.131]
  MoveL 1666 to (104.99, -64.77, 333.44) mm, rotated rx -20.49 ry -0.61 rz 0.23 deg; joints [-4.197, -123.194, -87.203, -50.32, 92.199, -9.408]
  MoveL 1667 to (105.13, -56.57, 331.13) mm, rotated rx -19.68 ry -0.66 rz 0.24 deg; joints [-4.417, -122.141, -89.676, -48.119, 92.425, -9.603]
  MoveL 1668 to (105.24, -52, 329) mm, rotated rx -19.2 ry -0.73 rz 0.26 deg; joints [-4.575, -121.471, -91.082, -46.925, 92.607, -9.744]
  MoveL 1669 to (104.83, -45.53, 326.37) mm, rotated rx -18.91 ry -0.84 rz 0.29 deg; joints [-4.721, -120.699, -92.661, -45.858, 92.793, -9.879]
  MoveL 1670 to (104.93, -34.87, 322.78) mm, rotated rx -18.74 ry -1.29 rz 0.44 deg; joints [-5.145, -119.722, -94.726, -44.706, 93.365, -10.295]
  MoveL 1671 to (105.81, -26.76, 320.85) mm, rotated rx -18.76 ry -1.56 rz 0.53 deg; joints [-5.497, -119.155, -96.065, -44.022, 93.711, -10.645]
  MoveL 1672 to (104.19, -21.96, 318.5) mm, rotated rx -19.09 ry -1.62 rz 0.56 deg; joints [-5.445, -118.674, -96.767, -44.133, 93.711, -10.607]
  MoveL 1673 to (104.96, -14.18, 316.45) mm, rotated rx -19.1 ry -1.79 rz 0.62 deg; joints [-5.738, -118.095, -98.083, -43.453, 93.932, -10.898]
  MoveL 1674 to (104.97, -4.46, 313.47) mm, rotated rx -18.9 ry -1.54 rz 0.53 deg; joints [-5.809, -117.147, -100.136, -42.116, 93.723, -10.957]
  MoveL 1675 to (106.32, 2.93, 310.37) mm, rotated rx -18.94 ry -1.33 rz 0.46 deg; joints [-5.97, -116.433, -101.462, -41.506, 93.528, -11.115]
  MoveL 1676 to (104.06, 6.88, 308.38) mm, rotated rx -19.01 ry -1.21 rz 0.42 deg; joints [-5.769, -115.908, -102.326, -41.202, 93.356, -10.918]
  MoveL 1677 to (105.14, 15.06, 306.55) mm, rotated rx -18.98 ry -1.19 rz 0.41 deg; joints [-6.016, -115.338, -103.713, -40.371, 93.381, -11.16]
  MoveL 1678 to (104.9, 25.12, 302.81) mm, rotated rx -18.52 ry -0.98 rz 0.33 deg; joints [-6.136, -114.252, -106.018, -38.659, 93.278, -11.258]
  MoveL 1679 to (105.04, 31.9, 300) mm, rotated rx -18.78 ry -0.73 rz 0.25 deg; joints [-6.129, -113.626, -107.07, -38.436, 92.965, -11.259]
  MoveL 1680 to (105.01, 36.45, 298.79) mm, rotated rx -18.86 ry -0.62 rz 0.21 deg; joints [-6.147, -113.28, -107.812, -38.105, 92.837, -11.278]
  MoveL 1681 to (105.02, 44.65, 296.47) mm, rotated rx -18.72 ry -0.53 rz 0.18 deg; joints [-6.287, -112.598, -109.359, -37.092, 92.803, -11.409]
  MoveL 1682 to (104.97, 54.84, 292.66) mm, rotated rx -18.32 ry -0.71 rz 0.24 deg; joints [-6.664, -111.647, -111.386, -35.681, 93.142, -11.766]
  MoveL 1683 to (105.13, 62.77, 290.48) mm, rotated rx -18.2 ry -0.91 rz 0.3 deg; joints [-6.99, -111.086, -112.722, -34.841, 93.433, -12.084]
  MoveL 1684 to (104.91, 67.51, 288.55) mm, rotated rx -18.03 ry -0.89 rz 0.29 deg; joints [-7.093, -110.609, -113.686, -34.191, 93.467, -12.177]
  MoveL 1685 to (104.99, 74.6, 286.11) mm, rotated rx -17.95 ry -0.89 rz 0.29 deg; joints [-7.29, -110.022, -114.917, -33.479, 93.527, -12.368]
  MoveL 1686 to (104.99, 84.79, 283.09) mm, rotated rx -17.86 ry -0.71 rz 0.23 deg; joints [-7.447, -109.224, -116.701, -32.381, 93.393, -12.515]
  MoveL 1687 to (105.03, 92.76, 280.75) mm, rotated rx -17.77 ry -0.66 rz 0.21 deg; joints [-7.634, -108.623, -118.076, -31.508, 93.392, -12.693]
  MoveL 1688 to (104.86, 97.37, 278.68) mm, rotated rx -17.76 ry -0.62 rz 0.2 deg; joints [-7.725, -108.177, -118.854, -31.173, 93.376, -12.782]
  MoveL 1689 to (105.05, 102.97, 277.03) mm, rotated rx -18.16 ry -0.71 rz 0.23 deg; joints [-7.898, -107.875, -119.361, -31.389, 93.412, -12.971]
  MoveL 1690 to (115.72, -262.51, 412) mm, rotated rx -18.32 ry -3.7 rz 1.22 deg; joints [-3.838, -153.298, -27.952, -77.779, 95.7, -9.027]
  MoveL 1691 to (115.08, -256, 411) mm, rotated rx -19.38 ry -3.4 rz 1.2 deg; joints [-3.701, -152.862, -28.751, -78.412, 95.219, -8.918]
  MoveL 1692 to (114.88, -250.47, 409) mm, rotated rx -20.34 ry -3.07 rz 1.14 deg; joints [-3.582, -152.416, -29.422, -79.077, 94.727, -8.82]
  MoveL 1693 to (114.96, -244.94, 406.79) mm, rotated rx -21.38 ry -2.68 rz 1.05 deg; joints [-3.451, -152.06, -29.87, -79.946, 94.15, -8.71]
  MoveL 1694 to (115.06, -234.99, 402.16) mm, rotated rx -23.08 ry -2.54 rz 1.08 deg; joints [-3.441, -151.379, -30.765, -81.396, 93.782, -8.731]
  MoveL 1695 to (115.1, -224.63, 397.2) mm, rotated rx -23.37 ry -2.35 rz 1.02 deg; joints [-3.474, -148.941, -35.53, -79.336, 93.541, -8.767]
  MoveL 1696 to (114.86, -214.91, 393.36) mm, rotated rx -22.48 ry -2.24 rz 0.93 deg; joints [-3.566, -145.886, -41.909, -75.117, 93.551, -8.841]
  MoveL 1697 to (115.3, -206.71, 390.77) mm, rotated rx -22.03 ry -2.14 rz 0.87 deg; joints [-3.671, -143.981, -45.951, -72.522, 93.523, -8.936]
  MoveL 1698 to (114.14, -201.75, 388.58) mm, rotated rx -22.01 ry -1.86 rz 0.75 deg; joints [-3.539, -142.906, -48.073, -71.411, 93.207, -8.802]
  MoveL 1699 to (115.04, -194.7, 385.35) mm, rotated rx -22.22 ry -1.82 rz 0.74 deg; joints [-3.658, -141.818, -50.147, -70.628, 93.147, -8.923]
  MoveL 1700 to (114.98, -185.53, 381) mm, rotated rx -22.53 ry -2.14 rz 0.89 deg; joints [-3.883, -140.514, -52.59, -69.859, 93.481, -9.156]
  MoveL 1701 to (114.88, -180.59, 379) mm, rotated rx -22.38 ry -2.17 rz 0.89 deg; joints [-3.953, -139.612, -54.421, -68.796, 93.536, -9.224]
  MoveL 1702 to (114.97, -174.92, 377.11) mm, rotated rx -22.14 ry -2.2 rz 0.89 deg; joints [-4.056, -138.611, -56.534, -67.451, 93.62, -9.321]
  MoveL 1703 to (115.1, -164.44, 373.5) mm, rotated rx -21.59 ry -2.14 rz 0.85 deg; joints [-4.201, -136.755, -60.455, -64.843, 93.652, -9.452]
  MoveL 1704 to (115.11, -155.98, 371) mm, rotated rx -21.46 ry -2.12 rz 0.83 deg; joints [-4.306, -135.567, -62.979, -63.382, 93.663, -9.553]
  MoveL 1705 to (114.41, -151.13, 368.64) mm, rotated rx -21.31 ry -2.01 rz 0.78 deg; joints [-4.284, -134.711, -64.643, -62.412, 93.565, -9.527]
  MoveL 1706 to (114.91, -144.56, 365.41) mm, rotated rx -21.05 ry -1.77 rz 0.68 deg; joints [-4.329, -133.582, -66.853, -61.035, 93.359, -9.563]
  MoveL 1707 to (115.56, -135.21, 361.03) mm, rotated rx -21.42 ry -1.35 rz 0.53 deg; joints [-4.308, -132.409, -68.961, -60.389, 92.858, -9.547]
  MoveL 1708 to (111.16, -131.65, 359) mm, rotated rx -21.51 ry -1.49 rz 0.59 deg; joints [-4.081, -131.785, -70.04, -60.043, 92.96, -9.325]
  MoveL 1709 to (114.95, -125.39, 357.82) mm, rotated rx -22.09 ry -0.94 rz 0.38 deg; joints [-4.168, -131.458, -70.751, -60.137, 92.292, -9.421]
  MoveL 1710 to (114.97, -115.06, 354) mm, rotated rx -22.06 ry -0.49 rz 0.2 deg; joints [-4.114, -130.092, -73.484, -58.668, 91.813, -9.363]
  MoveL 1711 to (115.66, -106.99, 350.54) mm, rotated rx -21.51 ry -0.57 rz 0.22 deg; joints [-4.355, -128.859, -76.02, -56.835, 92.018, -9.59]
  MoveL 1712 to (114.81, -101.87, 348) mm, rotated rx -21.33 ry -0.66 rz 0.26 deg; joints [-4.42, -128.097, -77.474, -55.984, 92.154, -9.65]
  MoveL 1713 to (115.02, -94.05, 344.93) mm, rotated rx -21.04 ry -0.87 rz 0.34 deg; joints [-4.671, -127.114, -79.485, -54.724, 92.465, -9.893]
  MoveL 1714 to (115.01, -84.21, 341.73) mm, rotated rx -20.87 ry -1.16 rz 0.44 deg; joints [-4.962, -126.059, -81.715, -53.45, 92.843, -10.179]
  MoveL 1715 to (115.05, -78.48, 340) mm, rotated rx -21.03 ry -1.2 rz 0.46 deg; joints [-5.059, -125.552, -82.746, -53.093, 92.872, -10.28]
  MoveL 1716 to (114.98, -73.43, 337.47) mm, rotated rx -21 ry -1.16 rz 0.45 deg; joints [-5.123, -124.907, -83.918, -52.53, 92.846, -10.342]
  MoveL 1717 to (114.84, -64.68, 333.45) mm, rotated rx -20.54 ry -1.1 rz 0.41 deg; joints [-5.266, -123.687, -86.329, -50.882, 92.879, -10.469]
  MoveL 1718 to (115.03, -57.35, 330.6) mm, rotated rx -19.71 ry -1.02 rz 0.36 deg; joints [-5.435, -122.587, -88.746, -48.735, 92.971, -10.61]
  MoveL 1719 to (115.6, -52.42, 328.93) mm, rotated rx -19.2 ry -0.92 rz 0.32 deg; joints [-5.564, -121.927, -90.25, -47.385, 92.982, -10.719]
  MoveL 1720 to (114.82, -45.56, 327.6) mm, rotated rx -18.51 ry -1.09 rz 0.36 deg; joints [-5.748, -121.148, -92.258, -45.51, 93.315, -10.878]
  MoveL 1721 to (115, -34.96, 323.79) mm, rotated rx -18.44 ry -1.53 rz 0.51 deg; joints [-6.186, -120.197, -94.204, -44.564, 93.873, -11.312]
  MoveL 1722 to (115.67, -25.68, 320.87) mm, rotated rx -18.68 ry -1.61 rz 0.54 deg; joints [-6.438, -119.478, -95.652, -44.102, 93.952, -11.569]
  MoveL 1723 to (113.68, -20.96, 319) mm, rotated rx -18.94 ry -1.65 rz 0.57 deg; joints [-6.351, -119.019, -96.42, -44.051, 93.935, -11.495]
  MoveL 1724 to (114.87, -14.34, 316.82) mm, rotated rx -19.15 ry -1.61 rz 0.56 deg; joints [-6.547, -118.524, -97.387, -43.789, 93.885, -11.695]
  MoveL 1725 to (114.94, -4.33, 313.25) mm, rotated rx -19.08 ry -1.48 rz 0.51 deg; joints [-6.696, -117.554, -99.354, -42.707, 93.788, -11.837]
  MoveL 1726 to (115.27, 4.85, 310.49) mm, rotated rx -19.21 ry -1.51 rz 0.53 deg; joints [-6.92, -116.838, -100.85, -42.08, 93.839, -12.064]
  MoveL 1727 to (113.62, 9.26, 309) mm, rotated rx -19.14 ry -1.4 rz 0.48 deg; joints [-6.803, -116.34, -101.863, -41.467, 93.711, -11.944]
  MoveL 1728 to (115.21, 15.02, 306.87) mm, rotated rx -19 ry -1.33 rz 0.46 deg; joints [-7.057, -115.826, -102.947, -40.76, 93.712, -12.188]
  MoveL 1729 to (115.07, 25.1, 303.26) mm, rotated rx -18.82 ry -1.2 rz 0.41 deg; joints [-7.223, -114.853, -104.956, -39.527, 93.653, -12.342]
  MoveL 1730 to (114.9, 32.3, 300.07) mm, rotated rx -19.09 ry -0.93 rz 0.32 deg; joints [-7.2, -114.149, -106.115, -39.273, 93.315, -12.326]
  MoveL 1731 to (115.07, 36.7, 298.72) mm, rotated rx -19.04 ry -0.85 rz 0.29 deg; joints [-7.273, -113.772, -106.932, -38.774, 93.25, -12.396]
  MoveL 1732 to (115.09, 44.77, 296.57) mm, rotated rx -18.81 ry -0.79 rz 0.27 deg; joints [-7.45, -113.103, -108.523, -37.621, 93.269, -12.56]
  MoveL 1733 to (115.18, 54.74, 292.78) mm, rotated rx -18.26 ry -0.71 rz 0.23 deg; joints [-7.724, -112.087, -110.727, -35.896, 93.353, -12.805]
  MoveL 1734 to (114.79, 61.84, 290.29) mm, rotated rx -18.16 ry -0.64 rz 0.21 deg; joints [-7.837, -111.445, -112.06, -35.093, 93.328, -12.91]
  MoveL 1735 to (114.94, 66.56, 288.61) mm, rotated rx -18.04 ry -0.61 rz 0.2 deg; joints [-7.971, -111.031, -112.945, -34.509, 93.348, -13.036]
  MoveL 1736 to (115, 74.56, 286.16) mm, rotated rx -17.98 ry -0.54 rz 0.18 deg; joints [-8.155, -110.407, -114.319, -33.699, 93.334, -13.213]
  MoveL 1737 to (115.22, 85.17, 284.12) mm, rotated rx -18.04 ry -0.36 rz 0.12 deg; joints [-8.325, -109.773, -116.002, -32.668, 93.163, -13.38]
  MoveL 1738 to (114.77, 93.54, 280.67) mm, rotated rx -17.75 ry -0.41 rz 0.13 deg; joints [-8.594, -108.977, -117.62, -31.589, 93.344, -13.631]
  MoveL 1739 to (115.52, 97.74, 278.61) mm, rotated rx -17.65 ry -0.38 rz 0.12 deg; joints [-8.803, -108.575, -118.346, -31.174, 93.376, -13.83]
  MoveL 1740 to (115.13, 104.27, 276.85) mm, rotated rx -17.58 ry -0.48 rz 0.15 deg; joints [-9.018, -108.135, -119.41, -30.519, 93.539, -14.038]
  MoveL 1741 to (125.18, -263.08, 412) mm, rotated rx -18.89 ry -2.58 rz 0.88 deg; joints [-4.014, -154.549, -25.204, -79.689, 94.484, -9.202]
  MoveL 1742 to (124.98, -255.04, 411.05) mm, rotated rx -20.18 ry -2.23 rz 0.82 deg; joints [-3.888, -154.049, -26.178, -80.431, 93.91, -9.109]
  MoveL 1743 to (125.21, -244.79, 406.93) mm, rotated rx -21.79 ry -2.08 rz 0.83 deg; joints [-3.882, -153.15, -27.608, -81.463, 93.517, -9.14]
  MoveL 1744 to (125.14, -235.44, 402.61) mm, rotated rx -22.98 ry -1.96 rz 0.83 deg; joints [-3.882, -151.94, -29.717, -81.732, 93.222, -9.163]
  MoveL 1745 to (124.2, -224.93, 397.21) mm, rotated rx -23.03 ry -2.42 rz 1.03 deg; joints [-4.121, -149.244, -35.026, -79.249, 93.733, -9.406]
  MoveL 1746 to (125.18, -215.71, 394.3) mm, rotated rx -22.53 ry -2.94 rz 1.22 deg; joints [-4.517, -147.013, -39.786, -76.343, 94.403, -9.797]
  MoveL 1747 to (124.98, -206.75, 391) mm, rotated rx -22.39 ry -2.78 rz 1.15 deg; joints [-4.564, -145.045, -43.825, -74.103, 94.268, -9.838]
  MoveL 1748 to (130.61, -201.62, 389) mm, rotated rx -22.52 ry -2.63 rz 1.09 deg; joints [-4.945, -144.466, -44.994, -73.647, 94.129, -10.219]
  MoveL 1749 to (124.83, -201.31, 388.4) mm, rotated rx -22.42 ry -2.61 rz 1.07 deg; joints [-4.554, -143.938, -45.978, -73.064, 94.073, -9.827]
  MoveL 1750 to (125.1, -195.06, 385.89) mm, rotated rx -22.15 ry -2.49 rz 1.01 deg; joints [-4.62, -142.576, -48.777, -71.342, 93.993, -9.886]
  MoveL 1751 to (125.41, -185.41, 381.59) mm, rotated rx -22.49 ry -2.32 rz 0.96 deg; joints [-4.684, -141.103, -51.579, -70.324, 93.769, -9.954]
  MoveL 1752 to (124.78, -180.59, 379) mm, rotated rx -22.44 ry -2.23 rz 0.92 deg; joints [-4.677, -140.15, -53.393, -69.4, 93.687, -9.945]
  MoveL 1753 to (125.03, -175.15, 377.88) mm, rotated rx -22.1 ry -2.27 rz 0.92 deg; joints [-4.795, -139.193, -55.545, -67.88, 93.794, -10.056]
  MoveL 1754 to (124.83, -165.52, 374.89) mm, rotated rx -21.58 ry -2.43 rz 0.96 deg; joints [-5.006, -137.53, -59.128, -65.486, 94.076, -10.255]
  MoveL 1755 to (124.83, -156.95, 370.84) mm, rotated rx -21.62 ry -2.4 rz 0.95 deg; joints [-5.118, -136.243, -61.58, -64.368, 94.056, -10.367]
  MoveL 1756 to (125.13, -151.41, 368.5) mm, rotated rx -21.77 ry -2.17 rz 0.87 deg; joints [-5.114, -135.495, -63.003, -63.797, 93.786, -10.364]
  MoveL 1757 to (125.01, -144.56, 365.29) mm, rotated rx -21.79 ry -1.67 rz 0.67 deg; joints [-4.993, -134.389, -65.1, -62.734, 93.227, -10.238]
  MoveL 1758 to (125.12, -134.43, 361.39) mm, rotated rx -21.87 ry -0.84 rz 0.34 deg; joints [-4.789, -132.914, -68.009, -61.22, 92.313, -10.03]
  MoveL 1759 to (128.4, -128.26, 360) mm, rotated rx -22.43 ry -0.49 rz 0.2 deg; joints [-4.926, -132.584, -68.701, -61.344, 91.856, -10.176]
  MoveL 1760 to (124.71, -124.57, 358.13) mm, rotated rx -22.59 ry -0.46 rz 0.19 deg; joints [-4.681, -131.988, -69.743, -61.046, 91.774, -9.937]
  MoveL 1761 to (125.07, -114.96, 354) mm, rotated rx -21.99 ry -0.59 rz 0.24 deg; joints [-4.947, -130.483, -72.818, -58.917, 92.04, -10.188]
  MoveL 1762 to (123.58, -107.08, 350.52) mm, rotated rx -21.56 ry -0.48 rz 0.19 deg; joints [-4.938, -129.194, -75.402, -57.177, 92.006, -10.168]
  MoveL 1763 to (125.88, -102.76, 347.89) mm, rotated rx -21.24 ry -0.44 rz 0.17 deg; joints [-5.196, -128.513, -76.696, -56.246, 92.053, -10.414]
  MoveL 1764 to (125.17, -94.31, 345.17) mm, rotated rx -20.53 ry -0.6 rz 0.23 deg; joints [-5.397, -127.289, -79.402, -54.104, 92.381, -10.594]
  MoveL 1765 to (124.98, -84.38, 342.13) mm, rotated rx -20.68 ry -0.96 rz 0.36 deg; joints [-5.691, -126.395, -81.252, -53.383, 92.778, -10.893]
  MoveL 1766 to (124.83, -78.48, 340) mm, rotated rx -20.98 ry -1.1 rz 0.42 deg; joints [-5.816, -125.904, -82.154, -53.298, 92.885, -11.026]
  MoveL 1767 to (125.01, -73.54, 337.52) mm, rotated rx -21.1 ry -1.05 rz 0.41 deg; joints [-5.89, -125.346, -83.119, -53.007, 92.828, -11.103]
  MoveL 1768 to (124.86, -64.87, 333.47) mm, rotated rx -20.75 ry -0.76 rz 0.29 deg; joints [-5.928, -124.117, -85.508, -51.44, 92.594, -11.127]
  MoveL 1769 to (125.32, -55.84, 330.77) mm, rotated rx -19.59 ry -0.65 rz 0.23 deg; joints [-6.169, -122.815, -88.567, -48.537, 92.736, -11.327]
  MoveL 1770 to (124.35, -50.51, 329) mm, rotated rx -18.78 ry -0.72 rz 0.25 deg; joints [-6.291, -121.995, -90.498, -46.654, 92.991, -11.418]
  MoveL 1771 to (125.07, -44.74, 327.59) mm, rotated rx -18.1 ry -0.73 rz 0.24 deg; joints [-6.522, -121.314, -92.242, -44.932, 93.175, -11.618]
  MoveL 1772 to (125.12, -34.98, 324.41) mm, rotated rx -18.11 ry -1 rz 0.33 deg; joints [-6.847, -120.475, -93.996, -44.104, 93.516, -11.941]
  MoveL 1773 to (125.08, -24.69, 320.74) mm, rotated rx -18.96 ry -0.89 rz 0.3 deg; joints [-6.911, -119.736, -95.18, -44.468, 93.239, -12.037]
  MoveL 1774 to (124.59, -18.66, 320) mm, rotated rx -19.08 ry -0.8 rz 0.28 deg; joints [-6.922, -119.341, -96.205, -43.944, 93.129, -12.051]
  MoveL 1775 to (125, -13.76, 317.35) mm, rotated rx -19.12 ry -0.76 rz 0.26 deg; joints [-7.046, -118.795, -97.116, -43.61, 93.103, -12.174]
  MoveL 1776 to (124.96, -4.3, 313.04) mm, rotated rx -18.92 ry -1.04 rz 0.36 deg; joints [-7.417, -117.807, -98.988, -42.614, 93.499, -12.535]
  MoveL 1777 to (124.76, 3.83, 310.5) mm, rotated rx -19.12 ry -1.25 rz 0.43 deg; joints [-7.661, -117.207, -100.198, -42.268, 93.713, -12.787]
  MoveL 1778 to (125.66, 8.47, 308.67) mm, rotated rx -19.39 ry -1.24 rz 0.44 deg; joints [-7.821, -116.88, -100.734, -42.327, 93.68, -12.955]
  MoveL 1779 to (125.13, 14.92, 306.81) mm, rotated rx -19.16 ry -1.22 rz 0.42 deg; joints [-7.929, -116.266, -102.133, -41.319, 93.726, -13.052]
  MoveL 1780 to (125.22, 25.14, 303.56) mm, rotated rx -19.13 ry -0.84 rz 0.29 deg; joints [-7.972, -115.329, -104.1, -40.176, 93.345, -13.087]
  MoveL 1781 to (124.62, 32.96, 300.31) mm, rotated rx -19.11 ry -0.84 rz 0.29 deg; joints [-8.114, -114.559, -105.543, -39.493, 93.382, -13.227]
  MoveL 1782 to (125.64, 37.19, 298.76) mm, rotated rx -19.08 ry -0.99 rz 0.34 deg; joints [-8.404, -114.254, -106.178, -39.179, 93.594, -13.514]
  MoveL 1783 to (125.07, 44.61, 296.24) mm, rotated rx -18.86 ry -0.96 rz 0.33 deg; joints [-8.547, -113.55, -107.694, -38.156, 93.642, -13.644]
  MoveL 1784 to (124.91, 54.87, 292.64) mm, rotated rx -18.5 ry -1 rz 0.34 deg; joints [-8.869, -112.61, -109.738, -36.732, 93.827, -13.946]
  MoveL 1785 to (125.58, 63.07, 290.67) mm, rotated rx -18.3 ry -0.83 rz 0.27 deg; joints [-9.075, -112.008, -111.266, -35.585, 93.732, -14.136]
  MoveL 1786 to (124.08, 67.53, 288.79) mm, rotated rx -18.16 ry -0.63 rz 0.21 deg; joints [-8.951, -111.463, -112.321, -34.884, 93.541, -14.005]
  MoveL 1787 to (125.23, 74.99, 286.48) mm, rotated rx -18.18 ry -0.52 rz 0.17 deg; joints [-9.213, -110.936, -113.48, -34.255, 93.479, -14.261]
  MoveL 1788 to (124.75, 85.19, 283.3) mm, rotated rx -17.96 ry -0.43 rz 0.14 deg; joints [-9.429, -110.096, -115.378, -32.972, 93.48, -14.46]
  MoveL 1789 to (124.93, 92.94, 280.58) mm, rotated rx -17.41 ry -0.52 rz 0.16 deg; joints [-9.817, -109.423, -117.019, -31.52, 93.782, -14.813]
  MoveL 1790 to (124.96, 97.42, 278.82) mm, rotated rx -17.29 ry -0.55 rz 0.17 deg; joints [-10.001, -109.038, -117.823, -31.001, 93.885, -14.988]
  MoveL 1791 to (125, 104.54, 276.6) mm, rotated rx -17.25 ry -0.56 rz 0.17 deg; joints [-10.242, -108.532, -118.954, -30.361, 93.956, -15.223]
  MoveL 1792 to (125.92, 111.45, 276.16) mm, rotated rx -16.85 ry -0.7 rz 0.21 deg; joints [-10.698, -108.323, -120.155, -29.055, 94.299, -15.649]
  MoveL 1793 to (135.01, -263.47, 412.88) mm, rotated rx -18.95 ry -1.57 rz 0.54 deg; joints [-4.273, -155.294, -23.79, -80.273, 93.463, -9.447]
  MoveL 1794 to (134.79, -255.17, 411.71) mm, rotated rx -20.23 ry -1.91 rz 0.7 deg; joints [-4.4, -154.985, -24.378, -81.323, 93.644, -9.613]
  MoveL 1795 to (135.26, -244.2, 407.29) mm, rotated rx -22.06 ry -2.11 rz 0.86 deg; joints [-4.54, -154.351, -25.226, -82.961, 93.6, -9.799]
  MoveL 1796 to (134.77, -234.87, 403.96) mm, rotated rx -23.03 ry -1.7 rz 0.72 deg; joints [-4.411, -152.714, -28.393, -82.308, 92.995, -9.687]
  MoveL 1797 to (135.75, -228.04, 400.71) mm, rotated rx -22.76 ry -1.56 rz 0.66 deg; joints [-4.523, -150.476, -32.943, -79.712, 92.902, -9.792]
  MoveL 1798 to (134.86, -223.2, 397.82) mm, rotated rx -22.27 ry -1.71 rz 0.7 deg; joints [-4.614, -148.653, -36.621, -77.409, 93.148, -9.873]
  MoveL 1799 to (134.86, -215.47, 394.11) mm, rotated rx -22.29 ry -2 rz 0.82 deg; joints [-4.824, -147.005, -39.873, -75.885, 93.477, -10.086]
  MoveL 1800 to (135.03, -205.92, 391.2) mm, rotated rx -22.32 ry -2.37 rz 0.97 deg; joints [-5.096, -145.344, -43.358, -74.168, 93.9, -10.361]
  MoveL 1801 to (134.89, -195.4, 386.68) mm, rotated rx -22.32 ry -2.73 rz 1.12 deg; joints [-5.374, -143.453, -47.131, -72.373, 94.323, -10.642]
  MoveL 1802 to (135.01, -184.81, 381.62) mm, rotated rx -22.73 ry -2.43 rz 1.02 deg; joints [-5.391, -141.75, -50.324, -71.238, 93.937, -10.665]
  MoveL 1803 to (139.51, -179.08, 380) mm, rotated rx -22.92 ry -2.04 rz 0.86 deg; joints [-5.614, -141.141, -51.615, -70.689, 93.517, -10.886]
  MoveL 1804 to (134.83, -175.25, 378.32) mm, rotated rx -22.16 ry -1.98 rz 0.81 deg; joints [-5.366, -139.707, -54.617, -68.341, 93.552, -10.621]
  MoveL 1805 to (135, -165.5, 374.02) mm, rotated rx -21.6 ry -1.86 rz 0.74 deg; joints [-5.508, -137.786, -58.533, -65.777, 93.537, -10.747]
  MoveL 1806 to (134.12, -158.03, 370.45) mm, rotated rx -21.82 ry -1.81 rz 0.72 deg; joints [-5.521, -136.712, -60.517, -65.078, 93.441, -10.764]
  MoveL 1807 to (135.05, -152.83, 368.45) mm, rotated rx -22.33 ry -1.51 rz 0.62 deg; joints [-5.509, -136.252, -61.316, -65.18, 93.041, -10.762]
  MoveL 1808 to (135.23, -145.07, 365.98) mm, rotated rx -22.49 ry -1.16 rz 0.48 deg; joints [-5.473, -135.247, -63.361, -64.227, 92.628, -10.726]
  MoveL 1809 to (135.1, -134.63, 361.83) mm, rotated rx -22.39 ry -0.92 rz 0.38 deg; joints [-5.53, -133.718, -66.411, -62.567, 92.407, -10.779]
  MoveL 1810 to (133.11, -128.26, 360) mm, rotated rx -22.58 ry -0.68 rz 0.28 deg; joints [-5.352, -132.914, -68.047, -61.868, 92.086, -10.604]
  MoveL 1811 to (135.48, -124.24, 357.84) mm, rotated rx -22.52 ry -0.73 rz 0.3 deg; joints [-5.625, -132.418, -68.972, -61.397, 92.191, -10.875]
  MoveL 1812 to (135.18, -114.78, 353.53) mm, rotated rx -22.28 ry -0.46 rz 0.19 deg; joints [-5.654, -130.962, -71.816, -59.721, 91.95, -10.895]
  MoveL 1813 to (138.56, -108.23, 350) mm, rotated rx -21.85 ry -0.19 rz 0.08 deg; joints [-5.944, -129.934, -73.833, -58.267, 91.787, -11.17]
  MoveL 1814 to (134.98, -104.08, 347.8) mm, rotated rx -21.21 ry -0.25 rz 0.1 deg; joints [-5.814, -128.933, -75.855, -56.628, 91.95, -11.024]
  MoveL 1815 to (134.72, -94.54, 345.61) mm, rotated rx -20.32 ry -0.47 rz 0.17 deg; joints [-6.111, -127.635, -78.927, -54.027, 92.394, -11.292]
  MoveL 1816 to (135.14, -84.46, 342.72) mm, rotated rx -20.35 ry -0.79 rz 0.29 deg; joints [-6.459, -126.718, -80.905, -53.08, 92.787, -11.64]
  MoveL 1817 to (135.96, -77.96, 340) mm, rotated rx -20.96 ry -1.01 rz 0.39 deg; joints [-6.691, -126.311, -81.498, -53.549, 92.93, -11.891]
  MoveL 1818 to (134.8, -73.24, 337.87) mm, rotated rx -21.44 ry -0.84 rz 0.33 deg; joints [-6.566, -125.872, -82.155, -53.765, 92.639, -11.78]
  MoveL 1819 to (135.02, -64.76, 334.18) mm, rotated rx -20.99 ry -0.57 rz 0.22 deg; joints [-6.656, -124.673, -84.571, -52.057, 92.454, -11.853]
  MoveL 1820 to (134.7, -56.07, 331.17) mm, rotated rx -19.6 ry -0.39 rz 0.14 deg; joints [-6.833, -123.215, -87.934, -48.751, 92.577, -11.979]
  MoveL 1821 to (135.19, -50.9, 329) mm, rotated rx -18.9 ry -0.35 rz 0.12 deg; joints [-7.026, -122.432, -89.684, -47.103, 92.715, -12.141]
  MoveL 1822 to (135.19, -44.98, 327.27) mm, rotated rx -18.24 ry -0.19 rz 0.06 deg; joints [-7.129, -121.648, -91.564, -45.331, 92.712, -12.214]
  MoveL 1823 to (135.08, -35.08, 324.13) mm, rotated rx -18.06 ry -0.01 rz 0 deg; joints [-7.247, -120.647, -93.729, -43.95, 92.589, -12.32]
  MoveL 1824 to (134.82, -25.22, 320.97) mm, rotated rx -18.79 ry -0.23 rz 0.08 deg; joints [-7.459, -120.014, -94.814, -44.271, 92.697, -12.561]
  MoveL 1825 to (135.46, -20.27, 319) mm, rotated rx -18.94 ry -0.38 rz 0.13 deg; joints [-7.686, -119.633, -95.5, -44.162, 92.867, -12.792]
  MoveL 1826 to (134.85, -14.32, 317.39) mm, rotated rx -19.02 ry -0.52 rz 0.18 deg; joints [-7.815, -119.167, -96.506, -43.74, 93.012, -12.924]
  MoveL 1827 to (134.88, -4.39, 313) mm, rotated rx -18.77 ry -0.5 rz 0.17 deg; joints [-8.067, -118.077, -98.622, -42.475, 93.094, -13.161]
  MoveL 1828 to (134.91, 3.03, 310.68) mm, rotated rx -19.07 ry -0.59 rz 0.2 deg; joints [-8.251, -117.552, -99.638, -42.312, 93.156, -13.357]
  MoveL 1829 to (134.99, 7.8, 308.4) mm, rotated rx -19.24 ry -0.65 rz 0.23 deg; joints [-8.386, -117.115, -100.34, -42.232, 93.197, -13.498]
  MoveL 1830 to (135.15, 15, 307.08) mm, rotated rx -19.37 ry -0.67 rz 0.24 deg; joints [-8.558, -116.677, -101.438, -41.716, 93.224, -13.673]
  MoveL 1831 to (135.05, 25.17, 303.62) mm, rotated rx -19.15 ry -0.75 rz 0.26 deg; joints [-8.866, -115.757, -103.406, -40.491, 93.409, -13.969]
  MoveL 1832 to (135.81, 33.46, 300.43) mm, rotated rx -18.79 ry -0.84 rz 0.29 deg; joints [-9.253, -114.973, -105.086, -39.295, 93.665, -14.335]
  MoveL 1833 to (133.8, 37.45, 298.68) mm, rotated rx -18.88 ry -0.96 rz 0.33 deg; joints [-9.216, -114.543, -105.816, -39.102, 93.751, -14.305]
  MoveL 1834 to (135.08, 44.74, 296.85) mm, rotated rx -18.69 ry -1.19 rz 0.4 deg; joints [-9.682, -114.086, -107.011, -38.27, 94.12, -14.759]
  MoveL 1835 to (134.96, 54.94, 293.2) mm, rotated rx -18.55 ry -1.49 rz 0.5 deg; joints [-10.145, -113.265, -108.728, -37.36, 94.549, -15.214]
  MoveL 1836 to (134.8, 63.11, 290.81) mm, rotated rx -18.61 ry -1.3 rz 0.44 deg; joints [-10.245, -112.624, -110.112, -36.632, 94.358, -15.312]
  MoveL 1837 to (135.22, 67.9, 288.78) mm, rotated rx -18.45 ry -1.17 rz 0.39 deg; joints [-10.388, -112.146, -111.076, -35.96, 94.3, -15.442]
  MoveL 1838 to (135.25, 74.92, 286.51) mm, rotated rx -18.31 ry -1.04 rz 0.35 deg; joints [-10.547, -111.554, -112.387, -35.083, 94.233, -15.589]
  MoveL 1839 to (134.88, 85.12, 283.22) mm, rotated rx -17.86 ry -0.92 rz 0.3 deg; joints [-10.821, -110.66, -114.474, -33.447, 94.282, -15.831]
  MoveL 1840 to (134.67, 92.38, 280.65) mm, rotated rx -17.43 ry -0.86 rz 0.27 deg; joints [-11.07, -109.998, -116.027, -32.138, 94.39, -16.05]
  MoveL 1841 to (135.02, 96.87, 278.57) mm, rotated rx -17.22 ry -0.82 rz 0.26 deg; joints [-11.275, -109.558, -116.911, -31.496, 94.448, -16.239]
  MoveL 1842 to (134.85, 104.66, 276.57) mm, rotated rx -17.03 ry -0.99 rz 0.3 deg; joints [-11.644, -109.073, -118.198, -30.59, 94.742, -16.593]
  MoveL 1843 to (135.81, 113.19, 275.37) mm, rotated rx -16.74 ry -1.02 rz 0.31 deg; joints [-12.099, -108.719, -119.601, -29.303, 94.958, -17.021]
  MoveL 1844 to (141.93, -261.81, 414.25) mm, rotated rx -19.35 ry -2.18 rz 0.76 deg; joints [-4.928, -156.753, -21.014, -82.127, 94.155, -10.112]
  MoveL 1845 to (142.81, -254.77, 412.27) mm, rotated rx -20.25 ry -2.03 rz 0.75 deg; joints [-4.965, -155.851, -22.743, -82.163, 93.863, -10.173]
  MoveL 1846 to (144.49, -243.48, 406.17) mm, rotated rx -22.65 ry -1.46 rz 0.61 deg; joints [-4.877, -155.499, -22.669, -84.856, 92.855, -10.141]
  MoveL 1847 to (145.09, -235.6, 404) mm, rotated rx -23.53 ry -0.95 rz 0.42 deg; joints [-4.767, -154.177, -25.313, -84.304, 92.152, -10.045]
  MoveL 1848 to (145.24, -227.76, 401.13) mm, rotated rx -22.88 ry -0.72 rz 0.3 deg; joints [-4.822, -150.98, -32.012, -80.119, 92.012, -10.085]
  MoveL 1849 to (145.33, -221.81, 397.95) mm, rotated rx -21.94 ry -0.64 rz 0.26 deg; joints [-4.937, -148.39, -37.382, -76.402, 92.108, -10.178]
  MoveL 1850 to (145.41, -214.18, 395.11) mm, rotated rx -21.62 ry -1 rz 0.4 deg; joints [-5.198, -146.616, -41.086, -74.234, 92.577, -10.43]
  MoveL 1851 to (144.99, -205.13, 392.15) mm, rotated rx -21.42 ry -1.91 rz 0.75 deg; joints [-5.654, -145.026, -44.447, -72.466, 93.642, -10.887]
  MoveL 1852 to (144.58, -195, 386.76) mm, rotated rx -22.33 ry -2.5 rz 1.03 deg; joints [-5.95, -143.91, -46.296, -72.764, 94.148, -11.213]
  MoveL 1853 to (144.94, -185.15, 382.22) mm, rotated rx -23.18 ry -2.03 rz 0.87 deg; joints [-5.882, -142.639, -48.555, -72.519, 93.487, -11.158]
  MoveL 1854 to (145.54, -178.36, 380.33) mm, rotated rx -23.03 ry -1.83 rz 0.78 deg; joints [-5.947, -141.438, -51.12, -70.974, 93.307, -11.217]
  MoveL 1855 to (144.51, -173.72, 378.55) mm, rotated rx -22.56 ry -1.62 rz 0.67 deg; joints [-5.892, -140.235, -53.64, -69.145, 93.166, -11.149]
  MoveL 1856 to (145.05, -165.55, 374.24) mm, rotated rx -21.99 ry -1.04 rz 0.42 deg; joints [-5.863, -138.346, -57.402, -66.597, 92.645, -11.1]
  MoveL 1857 to (145.78, -156.32, 370.77) mm, rotated rx -21.96 ry -0.94 rz 0.38 deg; joints [-6.017, -137.004, -60.122, -65.173, 92.569, -11.251]
  MoveL 1858 to (142.87, -152.29, 368.67) mm, rotated rx -22.31 ry -0.99 rz 0.41 deg; joints [-5.866, -136.453, -61.034, -65.158, 92.535, -11.111]
  MoveL 1859 to (148.89, -149.23, 370) mm, rotated rx -22.17 ry -1.41 rz 0.58 deg; joints [-6.517, -136.626, -61.159, -64.843, 93.093, -11.758]
  MoveL 1860 to (144.74, -144.69, 366.5) mm, rotated rx -22.34 ry -1.44 rz 0.59 deg; joints [-6.301, -135.709, -62.654, -64.427, 93.065, -11.548]
  MoveL 1861 to (145.21, -135.32, 362.07) mm, rotated rx -22.51 ry -1.43 rz 0.59 deg; joints [-6.473, -134.468, -64.971, -63.521, 93.036, -11.723]
  MoveL 1862 to (144.69, -125.23, 357.46) mm, rotated rx -22.96 ry -1.26 rz 0.53 deg; joints [-6.5, -133.249, -67.174, -62.945, 92.776, -11.759]
  MoveL 1863 to (144.92, -114.85, 352.93) mm, rotated rx -22.8 ry -0.66 rz 0.28 deg; joints [-6.446, -131.651, -70.303, -61.126, 92.157, -11.696]
  MoveL 1864 to (145.35, -107.19, 350.14) mm, rotated rx -21.76 ry -0.56 rz 0.23 deg; joints [-6.653, -130.214, -73.448, -58.39, 92.294, -11.873]
  MoveL 1865 to (144.93, -102.27, 348.6) mm, rotated rx -20.85 ry -0.57 rz 0.22 deg; joints [-6.783, -129.228, -75.712, -56.223, 92.5, -11.974]
  MoveL 1866 to (144.9, -94.21, 345.51) mm, rotated rx -19.95 ry -0.74 rz 0.27 deg; joints [-7.081, -127.95, -78.515, -53.869, 92.91, -12.24]
  MoveL 1867 to (144.85, -84.35, 342.19) mm, rotated rx -20.08 ry -0.93 rz 0.34 deg; joints [-7.335, -126.998, -80.441, -53.08, 93.13, -12.497]
  MoveL 1868 to (144.53, -77.88, 340.12) mm, rotated rx -21.06 ry -0.88 rz 0.34 deg; joints [-7.316, -126.709, -80.789, -53.965, 92.869, -12.512]
  MoveL 1869 to (145.39, -73.22, 338.03) mm, rotated rx -21.56 ry -0.79 rz 0.31 deg; joints [-7.39, -126.391, -81.23, -54.315, 92.677, -12.599]
  MoveL 1870 to (144.81, -64.96, 334.07) mm, rotated rx -21.14 ry -1.07 rz 0.41 deg; joints [-7.678, -125.271, -83.421, -52.914, 93.096, -12.875]
  MoveL 1871 to (144.76, -57.2, 331.11) mm, rotated rx -20.02 ry -0.87 rz 0.32 deg; joints [-7.85, -123.973, -86.322, -50.182, 93.164, -13.003]
  MoveL 1872 to (145.07, -52.59, 328.68) mm, rotated rx -19.49 ry -0.64 rz 0.23 deg; joints [-7.922, -123.189, -87.925, -48.79, 93.052, -13.051]
  MoveL 1873 to (144.84, -45.57, 327.01) mm, rotated rx -18.82 ry -0.3 rz 0.1 deg; joints [-7.947, -122.281, -90.127, -46.768, 92.852, -13.043]
  MoveL 1874 to (145, -34.94, 324.01) mm, rotated rx -18.13 ry 0.07 rz -0.02 deg; joints [-8.08, -121.06, -92.993, -44.362, 92.662, -13.138]
  MoveL 1875 to (144.66, -26.02, 320.92) mm, rotated rx -18.36 ry -0.14 rz 0.05 deg; joints [-8.323, -120.331, -94.4, -43.972, 92.872, -13.39]
  MoveL 1876 to (145.3, -21.01, 318.73) mm, rotated rx -18.75 ry -0.29 rz 0.1 deg; joints [-8.528, -119.991, -94.88, -44.254, 92.975, -13.611]
  MoveL 1877 to (144.96, -14.44, 317.01) mm, rotated rx -18.74 ry -0.53 rz 0.18 deg; joints [-8.76, -119.491, -96.016, -43.683, 93.259, -13.843]
  MoveL 1878 to (145.02, -4.39, 313.84) mm, rotated rx -18.82 ry -0.66 rz 0.23 deg; joints [-9.063, -118.679, -97.719, -42.92, 93.44, -14.146]
  MoveL 1879 to (145.59, 5.04, 311.18) mm, rotated rx -18.99 ry -0.72 rz 0.25 deg; joints [-9.346, -118.002, -99.181, -42.329, 93.506, -14.434]
  MoveL 1880 to (141.41, 8.43, 309) mm, rotated rx -19.25 ry -0.61 rz 0.21 deg; joints [-8.97, -117.444, -99.943, -42.338, 93.265, -14.073]
  MoveL 1881 to (145.18, 15.07, 307.35) mm, rotated rx -19.32 ry -0.74 rz 0.26 deg; joints [-9.538, -117.161, -100.705, -41.988, 93.483, -14.638]
  MoveL 1882 to (145.04, 25.15, 303.65) mm, rotated rx -18.97 ry -0.79 rz 0.27 deg; joints [-9.862, -116.181, -102.79, -40.583, 93.68, -14.943]
  MoveL 1883 to (144.55, 33.69, 300.39) mm, rotated rx -18.72 ry -0.85 rz 0.29 deg; joints [-10.114, -115.345, -104.524, -39.47, 93.847, -15.18]
  MoveL 1884 to (146.26, 37.68, 299) mm, rotated rx -18.49 ry -0.98 rz 0.33 deg; joints [-10.492, -115.065, -105.223, -38.891, 94.109, -15.543]
  MoveL 1885 to (144.91, 44.74, 297.36) mm, rotated rx -18.13 ry -1.36 rz 0.45 deg; joints [-10.813, -114.525, -106.644, -37.792, 94.655, -15.848]
  MoveL 1886 to (145.06, 55.15, 293.54) mm, rotated rx -18.39 ry -1.72 rz 0.57 deg; joints [-11.299, -113.798, -108.008, -37.543, 95.036, -16.349]
  MoveL 1887 to (145.39, 63.39, 290.58) mm, rotated rx -18.81 ry -1.82 rz 0.62 deg; joints [-11.585, -113.258, -108.934, -37.626, 95.079, -16.657]
  MoveL 1888 to (143.99, 68.02, 288.9) mm, rotated rx -18.73 ry -1.68 rz 0.57 deg; joints [-11.526, -112.76, -109.94, -36.992, 94.949, -16.591]
  MoveL 1889 to (144.98, 75.37, 286.23) mm, rotated rx -18.53 ry -1.43 rz 0.48 deg; joints [-11.752, -112.109, -111.348, -35.982, 94.789, -16.796]
  MoveL 1890 to (145.05, 85.62, 283.03) mm, rotated rx -18.05 ry -1.45 rz 0.47 deg; joints [-12.183, -111.277, -113.363, -34.383, 95.024, -17.195]
  MoveL 1891 to (145.25, 93.32, 280.54) mm, rotated rx -17.59 ry -1.23 rz 0.39 deg; joints [-12.417, -110.595, -115.029, -32.914, 94.982, -17.393]
  MoveL 1892 to (144.94, 97.74, 279) mm, rotated rx -17.4 ry -1.16 rz 0.36 deg; joints [-12.533, -110.198, -115.939, -32.2, 94.992, -17.493]
  MoveL 1893 to (144.93, 104.98, 277.45) mm, rotated rx -17.17 ry -1.17 rz 0.36 deg; joints [-12.827, -109.766, -117.209, -31.172, 95.133, -17.768]
  MoveL 1894 to (145.3, 114.89, 274.46) mm, rotated rx -17.03 ry -0.99 rz 0.3 deg; joints [-13.147, -109.066, -118.877, -30.042, 95.059, -18.068]
  MoveL 1895 to (148.03, 121.07, 273) mm, rotated rx -16.19 ry -0.7 rz 0.2 deg; joints [-13.662, -108.708, -120.351, -28.074, 95.142, -18.506]
  MoveL 1896 to (158.58, -252.08, 410.75) mm, rotated rx -21.69 ry -0.3 rz 0.12 deg; joints [-5.296, -158.211, -17.558, -86.11, 91.834, -10.525]
  MoveL 1897 to (155.51, -242.99, 406.5) mm, rotated rx -23.55 ry 0.07 rz -0.03 deg; joints [-4.967, -157.38, -18.751, -87.497, 91.067, -10.238]
  MoveL 1898 to (154.75, -234.86, 403.42) mm, rotated rx -23.63 ry 0.26 rz -0.11 deg; joints [-4.945, -154.326, -25.013, -84.334, 90.853, -10.218]
  MoveL 1899 to (153.84, -228.52, 400.5) mm, rotated rx -22.77 ry -0.03 rz 0.01 deg; joints [-5.129, -151.293, -31.326, -80.265, 91.332, -10.384]
  MoveL 1900 to (155, -223.36, 397.67) mm, rotated rx -21.87 ry -0.28 rz 0.11 deg; joints [-5.433, -149.097, -35.9, -77.063, 91.806, -10.665]
  MoveL 1901 to (155.11, -215.49, 395.4) mm, rotated rx -20.97 ry -0.8 rz 0.31 deg; joints [-5.8, -146.817, -40.867, -73.603, 92.572, -11.007]
  MoveL 1902 to (154.85, -205.18, 391.64) mm, rotated rx -20.54 ry -1.55 rz 0.58 deg; joints [-6.245, -144.734, -45.245, -71.063, 93.506, -11.443]
  MoveL 1903 to (155.74, -195.13, 387.73) mm, rotated rx -22.23 ry -1.69 rz 0.69 deg; joints [-6.392, -144.367, -45.582, -72.788, 93.357, -11.639]
  MoveL 1904 to (154.99, -185.29, 383.97) mm, rotated rx -23.5 ry -1.54 rz 0.67 deg; joints [-6.342, -143.541, -46.973, -73.436, 92.955, -11.617]
  MoveL 1905 to (153.38, -177.91, 380.33) mm, rotated rx -23.2 ry -1.6 rz 0.69 deg; joints [-6.394, -141.878, -50.273, -71.523, 93.083, -11.663]
  MoveL 1906 to (155.25, -173.65, 377.96) mm, rotated rx -22.8 ry -1.62 rz 0.68 deg; joints [-6.629, -140.911, -52.221, -70.159, 93.202, -11.888]
  MoveL 1907 to (155.07, -164.75, 374.68) mm, rotated rx -22.24 ry -1.75 rz 0.72 deg; joints [-6.851, -139.193, -55.836, -67.762, 93.479, -12.096]
  MoveL 1908 to (155.12, -154.69, 371.34) mm, rotated rx -21.92 ry -1.57 rz 0.63 deg; joints [-6.966, -137.52, -59.359, -65.559, 93.366, -12.199]
  MoveL 1909 to (152.76, -149.23, 370) mm, rotated rx -22.14 ry -1.52 rz 0.62 deg; joints [-6.844, -136.829, -60.792, -65.015, 93.256, -12.083]
  MoveL 1910 to (155.41, -144.57, 366.65) mm, rotated rx -22.38 ry -1.33 rz 0.55 deg; joints [-7.028, -136.24, -61.695, -64.912, 93.032, -12.27]
  MoveL 1911 to (155.09, -134.73, 362.31) mm, rotated rx -22.64 ry -1.07 rz 0.45 deg; joints [-7.045, -134.904, -64.219, -63.915, 92.704, -12.291]
  MoveL 1912 to (156.16, -128.26, 360) mm, rotated rx -22.96 ry -0.92 rz 0.39 deg; joints [-7.144, -134.261, -65.464, -63.599, 92.491, -12.396]
  MoveL 1913 to (154.72, -123.79, 357.32) mm, rotated rx -23.15 ry -0.97 rz 0.41 deg; joints [-7.126, -133.622, -66.533, -63.367, 92.498, -12.384]
  MoveL 1914 to (155.02, -115.01, 353.96) mm, rotated rx -22.96 ry -1.37 rz 0.58 deg; joints [-7.492, -132.516, -68.795, -62.13, 93.005, -12.747]
  MoveL 1915 to (154.87, -106.84, 350.91) mm, rotated rx -21.7 ry -1.7 rz 0.68 deg; joints [-7.884, -130.961, -72.228, -59.118, 93.671, -13.106]
  MoveL 1916 to (155.06, -101.72, 348.42) mm, rotated rx -20.77 ry -1.65 rz 0.63 deg; joints [-8.064, -129.855, -74.6, -56.942, 93.846, -13.253]
  MoveL 1917 to (155.01, -94.16, 345.11) mm, rotated rx -19.86 ry -1.32 rz 0.48 deg; joints [-8.152, -128.461, -77.565, -54.416, 93.716, -13.301]
  MoveL 1918 to (154.86, -84.5, 342.76) mm, rotated rx -20.4 ry -0.86 rz 0.32 deg; joints [-8.065, -127.643, -79.255, -53.956, 93.107, -13.23]
  MoveL 1919 to (155.9, -78.02, 340.07) mm, rotated rx -21.06 ry -0.86 rz 0.33 deg; joints [-8.215, -127.227, -79.861, -54.418, 92.98, -13.402]
  MoveL 1920 to (154.59, -73.36, 338.1) mm, rotated rx -21.25 ry -1.05 rz 0.41 deg; joints [-8.276, -126.758, -80.693, -54.288, 93.148, -13.472]
  MoveL 1921 to (154.89, -64.91, 334.48) mm, rotated rx -21.06 ry -1.36 rz 0.52 deg; joints [-8.641, -125.809, -82.568, -53.271, 93.564, -13.83]
  MoveL 1922 to (155.42, -56.81, 331.17) mm, rotated rx -20.4 ry -1.03 rz 0.38 deg; joints [-8.775, -124.615, -85.092, -51.222, 93.392, -13.934]
  MoveL 1923 to (154.43, -52.04, 328.95) mm, rotated rx -19.75 ry -0.89 rz 0.32 deg; joints [-8.805, -123.76, -86.903, -49.609, 93.401, -13.936]
  MoveL 1924 to (154.92, -45.36, 327.42) mm, rotated rx -18.98 ry -1.03 rz 0.35 deg; joints [-9.135, -122.983, -88.89, -47.7, 93.784, -14.23]
  MoveL 1925 to (155.05, -34.99, 323.94) mm, rotated rx -18.29 ry -1.12 rz 0.37 deg; joints [-9.507, -121.816, -91.537, -45.6, 94.116, -14.566]
  MoveL 1926 to (155.1, -25.33, 320.76) mm, rotated rx -18.15 ry -0.95 rz 0.31 deg; joints [-9.677, -120.863, -93.574, -44.347, 94.012, -14.723]
  MoveL 1927 to (153.47, -20.44, 319) mm, rotated rx -18.33 ry -0.9 rz 0.3 deg; joints [-9.609, -120.375, -94.472, -44.095, 93.907, -14.664]
  MoveL 1928 to (155.13, -14.31, 317.31) mm, rotated rx -18.54 ry -1.16 rz 0.39 deg; joints [-10.002, -120.066, -95.153, -44.018, 94.186, -15.066]
  MoveL 1929 to (155.12, -4.29, 314.05) mm, rotated rx -18.81 ry -1.09 rz 0.37 deg; joints [-10.186, -119.258, -96.759, -43.481, 94.08, -15.259]
  MoveL 1930 to (154.93, 5.25, 311.2) mm, rotated rx -19.15 ry -1.05 rz 0.36 deg; joints [-10.349, -118.549, -98.19, -43.086, 93.982, -15.435]
  MoveL 1931 to (158.67, 9.44, 309) mm, rotated rx -19.31 ry -1.05 rz 0.37 deg; joints [-10.787, -118.317, -98.52, -43.176, 94.014, -15.876]
  MoveL 1932 to (155.09, 14.96, 306.99) mm, rotated rx -19.27 ry -0.93 rz 0.32 deg; joints [-10.556, -117.614, -99.888, -42.422, 93.861, -15.643]
  MoveL 1933 to (154.92, 25.07, 303.38) mm, rotated rx -18.99 ry -0.76 rz 0.26 deg; joints [-10.774, -116.612, -102.021, -40.982, 93.807, -15.841]
  MoveL 1934 to (156.07, 34.32, 300.07) mm, rotated rx -18.3 ry -1.03 rz 0.34 deg; joints [-11.387, -115.769, -104.021, -39.28, 94.377, -16.415]
  MoveL 1935 to (152.38, 36.67, 299) mm, rotated rx -18.27 ry -1.09 rz 0.36 deg; joints [-11.145, -115.37, -104.725, -38.949, 94.402, -16.176]
  MoveL 1936 to (154.95, 44.97, 297.63) mm, rotated rx -17.76 ry -1.49 rz 0.48 deg; joints [-11.911, -114.985, -106.127, -37.622, 95.096, -16.912]
  MoveL 1937 to (155, 54.95, 293.66) mm, rotated rx -18.22 ry -1.71 rz 0.56 deg; joints [-12.29, -114.272, -107.312, -37.69, 95.262, -17.318]
  MoveL 1938 to (155.19, 64.87, 291.14) mm, rotated rx -18.98 ry -1.74 rz 0.6 deg; joints [-12.512, -113.787, -108.232, -38.02, 95.109, -17.58]
  MoveL 1939 to (151.8, 69.25, 289) mm, rotated rx -18.89 ry -1.67 rz 0.57 deg; joints [-12.309, -113.15, -109.366, -37.389, 95.033, -17.372]
  MoveL 1940 to (154.94, 74.71, 287.04) mm, rotated rx -18.58 ry -1.71 rz 0.57 deg; joints [-12.877, -112.817, -110.234, -36.622, 95.262, -17.918]
  MoveL 1941 to (155.06, 84.45, 283.9) mm, rotated rx -18.18 ry -1.68 rz 0.55 deg; joints [-13.276, -112.018, -112.122, -35.178, 95.423, -18.288]
  MoveL 1942 to (155.55, 94.11, 281.23) mm, rotated rx -17.85 ry -1.53 rz 0.49 deg; joints [-13.638, -111.313, -113.921, -33.754, 95.443, -18.62]
  MoveL 1943 to (152.44, 98.33, 279) mm, rotated rx -17.61 ry -1.36 rz 0.43 deg; joints [-13.426, -110.651, -115.139, -32.895, 95.304, -18.391]
  MoveL 1944 to (158.96, 101.12, 280) mm, rotated rx -17.61 ry -1.52 rz 0.48 deg; joints [-14.277, -111.1, -114.876, -32.84, 95.636, -19.234]
  MoveL 1945 to (154.73, 105.34, 277.83) mm, rotated rx -17.43 ry -1.31 rz 0.41 deg; joints [-13.92, -110.392, -116.156, -31.991, 95.417, -18.864]
  MoveL 1946 to (154.98, 115.17, 274.06) mm, rotated rx -16.82 ry -1.04 rz 0.31 deg; joints [-14.295, -109.501, -118.255, -30.145, 95.418, -19.182]
  MoveL 1947 to (156.23, 122.12, 272.34) mm, rotated rx -16.18 ry -0.61 rz 0.18 deg; joints [-14.571, -109.01, -119.865, -28.3, 95.263, -19.393]
  MoveL 1948 to (166.95, -260.51, 414.29) mm, rotated rx -20.45 ry -0.49 rz 0.18 deg; joints [-5.869, -161.131, -11.915, -87.675, 92.357, -11.057]
  MoveL 1949 to (165.65, -254.5, 412.71) mm, rotated rx -21.67 ry -0.49 rz 0.2 deg; joints [-5.782, -161.007, -11.979, -88.927, 92.114, -11.007]
  MoveL 1950 to (164.57, -248.91, 410.3) mm, rotated rx -23.14 ry -0.1 rz 0.04 deg; joints [-5.552, -161.451, -10.7, -91.125, 91.395, -10.812]
  MoveL 1951 to (165.32, -243.55, 408.14) mm, rotated rx -23.82 ry -0.05 rz 0.02 deg; joints [-5.608, -160.172, -13.2, -90.556, 91.221, -10.882]
  MoveL 1952 to (165.33, -234.17, 403) mm, rotated rx -23.1 ry -0.62 rz 0.27 deg; joints [-6.002, -154.8, -24.198, -84.36, 92.012, -11.262]
  MoveL 1953 to (165.04, -224.37, 397) mm, rotated rx -21.51 ry -1.04 rz 0.41 deg; joints [-6.402, -149.868, -34.336, -77.693, 92.815, -11.621]
  MoveL 1954 to (164.99, -215.89, 394.63) mm, rotated rx -20.51 ry -1.21 rz 0.45 deg; joints [-6.651, -147.177, -40.191, -73.593, 93.227, -11.84]
  MoveL 1955 to (165.49, -205.38, 391.61) mm, rotated rx -20.4 ry -1.31 rz 0.49 deg; joints [-6.883, -145.232, -44.33, -71.329, 93.387, -12.067]
  MoveL 1956 to (164.53, -194.54, 387.96) mm, rotated rx -22.57 ry -0.97 rz 0.4 deg; joints [-6.691, -144.897, -44.554, -73.479, 92.57, -11.937]
  MoveL 1957 to (164.81, -184.83, 384.74) mm, rotated rx -23.51 ry -0.89 rz 0.39 deg; joints [-6.752, -143.96, -46.326, -73.555, 92.296, -12.019]
  MoveL 1958 to (166.45, -179.22, 380.29) mm, rotated rx -23.06 ry -0.88 rz 0.37 deg; joints [-6.999, -142.463, -49.134, -71.812, 92.403, -12.254]
  MoveL 1959 to (165.01, -173.73, 377) mm, rotated rx -22.43 ry -1.06 rz 0.44 deg; joints [-7.119, -140.939, -52.174, -69.727, 92.743, -12.359]
  MoveL 1960 to (164.62, -164.81, 374.29) mm, rotated rx -22.21 ry -1.28 rz 0.52 deg; joints [-7.34, -139.518, -55.199, -67.963, 93.052, -12.574]
  MoveL 1961 to (165.2, -155.36, 370.89) mm, rotated rx -22.38 ry -0.99 rz 0.41 deg; joints [-7.406, -138.193, -57.866, -66.723, 92.717, -12.642]
  MoveL 1962 to (165.13, -150.75, 369) mm, rotated rx -22.45 ry -0.82 rz 0.34 deg; joints [-7.406, -137.508, -59.208, -66.097, 92.524, -12.642]
  MoveL 1963 to (164.85, -145.25, 367.08) mm, rotated rx -22.61 ry -0.69 rz 0.29 deg; joints [-7.41, -136.796, -60.627, -65.513, 92.348, -12.649]
  MoveL 1964 to (165.03, -134.83, 362.78) mm, rotated rx -22.64 ry -0.71 rz 0.3 deg; joints [-7.613, -135.372, -63.434, -64.178, 92.387, -12.852]
  MoveL 1965 to (165.91, -127.85, 360) mm, rotated rx -22.79 ry -1.01 rz 0.42 deg; joints [-7.917, -134.644, -64.853, -63.716, 92.711, -13.161]
  MoveL 1966 to (164.54, -123.74, 358.23) mm, rotated rx -22.71 ry -1.17 rz 0.49 deg; joints [-7.969, -134.019, -66.081, -63.08, 92.903, -13.212]
  MoveL 1967 to (164.77, -115.22, 354.8) mm, rotated rx -22.17 ry -1.81 rz 0.74 deg; joints [-8.468, -132.816, -68.606, -61.416, 93.757, -13.702]
  MoveL 1968 to (165.08, -107.61, 350.96) mm, rotated rx -21.6 ry -2.36 rz 0.93 deg; joints [-8.939, -131.653, -70.943, -59.85, 94.525, -14.163]
  MoveL 1969 to (164.7, -102.13, 347.91) mm, rotated rx -21.15 ry -2.38 rz 0.92 deg; joints [-9.083, -130.663, -72.883, -58.474, 94.668, -14.291]
  MoveL 1970 to (164.84, -93.95, 344.85) mm, rotated rx -20.55 ry -1.84 rz 0.69 deg; joints [-9.088, -129.316, -75.737, -56.249, 94.251, -14.263]
  MoveL 1971 to (165.12, -84.58, 343.38) mm, rotated rx -20.59 ry -1.48 rz 0.56 deg; joints [-9.122, -128.431, -77.837, -54.986, 93.868, -14.293]
  MoveL 1972 to (164.81, -77.73, 340.43) mm, rotated rx -20.61 ry -1.76 rz 0.66 deg; joints [-9.371, -127.701, -79.23, -54.433, 94.188, -14.545]
  MoveL 1973 to (165.3, -72.96, 338.42) mm, rotated rx -20.7 ry -2.08 rz 0.78 deg; joints [-9.65, -127.301, -79.979, -54.277, 94.537, -14.832]
  MoveL 1974 to (165.1, -65.14, 335.04) mm, rotated rx -21.27 ry -2.15 rz 0.84 deg; joints [-9.79, -126.657, -81.028, -54.456, 94.498, -14.993]
  MoveL 1975 to (165.38, -55.29, 331.4) mm, rotated rx -20.29 ry -2 rz 0.74 deg; joints [-10.079, -125.215, -84.203, -51.749, 94.63, -15.239]
  MoveL 1976 to (161.34, -50.72, 329) mm, rotated rx -19.51 ry -1.6 rz 0.57 deg; joints [-9.761, -124.092, -86.51, -49.681, 94.351, -14.883]
  MoveL 1977 to (167.3, -48.57, 330) mm, rotated rx -19.19 ry -2.22 rz 0.77 deg; joints [-10.612, -124.406, -86.4, -49.4, 95.221, -15.724]
  MoveL 1978 to (164.75, -44.34, 327.58) mm, rotated rx -18.71 ry -2.03 rz 0.69 deg; joints [-10.483, -123.556, -88.073, -48.054, 95.125, -15.568]
  MoveL 1979 to (165.04, -35.12, 323.78) mm, rotated rx -18.27 ry -2.22 rz 0.73 deg; joints [-10.884, -122.531, -90.221, -46.594, 95.499, -15.947]
  MoveL 1980 to (164.92, -24.54, 321.16) mm, rotated rx -18.54 ry -1.7 rz 0.57 deg; joints [-10.856, -121.628, -92.173, -45.659, 94.9, -15.92]
  MoveL 1981 to (164.92, -14.29, 317.12) mm, rotated rx -18.27 ry -1.42 rz 0.47 deg; joints [-11.03, -120.494, -94.501, -44.136, 94.72, -16.07]
  MoveL 1982 to (164.84, -4.44, 313.23) mm, rotated rx -19 ry -1.48 rz 0.51 deg; joints [-11.228, -119.78, -95.622, -44.465, 94.619, -16.305]
  MoveL 1983 to (165.22, 4.98, 311.21) mm, rotated rx -19.5 ry -1.17 rz 0.42 deg; joints [-11.283, -119.188, -96.92, -44.161, 94.176, -16.378]
  MoveL 1984 to (162.71, 9.44, 309) mm, rotated rx -19.47 ry -1.04 rz 0.37 deg; joints [-11.126, -118.553, -98.056, -43.571, 94.02, -16.217]
  MoveL 1985 to (165.11, 14.99, 307.21) mm, rotated rx -19.51 ry -0.88 rz 0.31 deg; joints [-11.411, -118.178, -98.881, -43.132, 93.898, -16.498]
  MoveL 1986 to (164.83, 25.11, 303.36) mm, rotated rx -18.87 ry -0.89 rz 0.31 deg; joints [-11.781, -117.09, -101.27, -41.247, 94.157, -16.831]
  MoveL 1987 to (164.73, 34.14, 300.17) mm, rotated rx -17.91 ry -1.3 rz 0.42 deg; joints [-12.4, -116.189, -103.49, -39.183, 94.958, -17.397]
  MoveL 1988 to (166.08, 38.39, 299) mm, rotated rx -17.55 ry -1.56 rz 0.49 deg; joints [-12.85, -115.929, -104.276, -38.434, 95.416, -17.826]
  MoveL 1989 to (164.87, 44.8, 297.52) mm, rotated rx -17.45 ry -1.6 rz 0.5 deg; joints [-12.968, -115.431, -105.499, -37.631, 95.507, -17.936]
  MoveL 1990 to (165.1, 55.21, 294.63) mm, rotated rx -17.89 ry -2.03 rz 0.66 deg; joints [-13.484, -114.907, -106.596, -37.674, 95.905, -18.487]
  MoveL 1991 to (164.92, 65.14, 291) mm, rotated rx -18.82 ry -2.29 rz 0.78 deg; joints [-13.799, -114.357, -107.339, -38.482, 95.937, -18.862]
  MoveL 1992 to (168.79, 69.25, 289) mm, rotated rx -18.95 ry -2.33 rz 0.8 deg; joints [-14.324, -114.205, -107.558, -38.61, 96.018, -19.391]
  MoveL 1993 to (165.07, 74.96, 287.58) mm, rotated rx -18.7 ry -2.1 rz 0.71 deg; joints [-14.076, -113.527, -109.107, -37.398, 95.827, -19.123]
  MoveL 1994 to (165.04, 84.57, 284.27) mm, rotated rx -18.32 ry -1.78 rz 0.59 deg; joints [-14.313, -112.638, -111.111, -35.834, 95.67, -19.323]
  MoveL 1995 to (164.92, 94.41, 281.47) mm, rotated rx -18.05 ry -1.74 rz 0.57 deg; joints [-14.691, -111.919, -112.888, -34.541, 95.79, -19.679]
  MoveL 1996 to (168.06, 98.94, 279) mm, rotated rx -17.78 ry -1.72 rz 0.55 deg; joints [-15.24, -111.584, -113.566, -33.996, 95.954, -20.203]
  MoveL 1997 to (161.89, 100.76, 280) mm, rotated rx -17.62 ry -1.57 rz 0.5 deg; joints [-14.595, -111.279, -114.535, -33.063, 95.741, -19.55]
  MoveL 1998 to (165.21, 105.07, 277.49) mm, rotated rx -17.51 ry -1.51 rz 0.48 deg; joints [-15.117, -110.974, -115.059, -32.767, 95.821, -20.056]
  MoveL 1999 to (164.94, 115.12, 274.12) mm, rotated rx -17.08 ry -1.26 rz 0.39 deg; joints [-15.437, -110.137, -117.063, -31.139, 95.779, -20.331]
  MoveL 2000 to (165.46, 123.45, 271.96) mm, rotated rx -16.59 ry -1.04 rz 0.31 deg; joints [-15.808, -109.579, -118.722, -29.535, 95.813, -20.652]
  MoveL 2001 to (175.25, -262.78, 414.25) mm, rotated rx -18.97 ry -0.84 rz 0.29 deg; joints [-6.592, -159.907, -14.752, -84.715, 93.125, -11.723]
  MoveL 2002 to (174.99, -255.42, 411.81) mm, rotated rx -20.94 ry -1.04 rz 0.4 deg; joints [-6.618, -161.539, -10.94, -88.872, 92.957, -11.819]
  MoveL 2003 to (176.35, -250.47, 409) mm, rotated rx -22.02 ry -1.43 rz 0.58 deg; joints [-6.849, -162.537, -8.516, -91.453, 93.187, -12.084]
  MoveL 2004 to (174.65, -244.11, 407.24) mm, rotated rx -22.78 ry -1.84 rz 0.77 deg; joints [-6.926, -160.854, -11.925, -90.561, 93.478, -12.185]
  MoveL 2005 to (174.95, -234, 402.58) mm, rotated rx -22.56 ry -2.33 rz 0.97 deg; joints [-7.295, -155.927, -22.037, -85.292, 94.084, -12.554]
  MoveL 2006 to (174.93, -224.12, 397.46) mm, rotated rx -21.51 ry -2.48 rz 0.98 deg; joints [-7.583, -151.349, -31.481, -79.449, 94.484, -12.814]
  MoveL 2007 to (174.83, -214.86, 395) mm, rotated rx -20.75 ry -2.07 rz 0.78 deg; joints [-7.621, -148.332, -37.971, -75.148, 94.221, -12.82]
  MoveL 2008 to (175.11, -204.44, 392.44) mm, rotated rx -20.92 ry -1.29 rz 0.49 deg; joints [-7.487, -146.263, -42.345, -72.822, 93.345, -12.681]
  MoveL 2009 to (175.29, -198.06, 390) mm, rotated rx -22.26 ry -0.79 rz 0.32 deg; joints [-7.31, -146.025, -42.513, -74.078, 92.521, -12.541]
  MoveL 2010 to (174.92, -193.89, 387.96) mm, rotated rx -23.02 ry -0.56 rz 0.24 deg; joints [-7.207, -145.727, -42.885, -74.69, 92.103, -12.457]
  MoveL 2011 to (174.87, -186.05, 384.16) mm, rotated rx -23.36 ry -0.4 rz 0.17 deg; joints [-7.244, -144.401, -45.392, -73.807, 91.86, -12.501]
  MoveL 2012 to (175.81, -178.64, 380.47) mm, rotated rx -22.92 ry -0.61 rz 0.26 deg; joints [-7.555, -142.782, -48.657, -71.788, 92.219, -12.8]
  MoveL 2013 to (175.08, -173.75, 378.23) mm, rotated rx -22.43 ry -0.7 rz 0.29 deg; joints [-7.664, -141.556, -51.188, -70.036, 92.433, -12.896]
  MoveL 2014 to (174.93, -165.1, 374.88) mm, rotated rx -22.15 ry -0.66 rz 0.27 deg; joints [-7.807, -139.97, -54.458, -68.068, 92.465, -13.03]
  MoveL 2015 to (174.9, -155.04, 371.44) mm, rotated rx -22.76 ry -0.43 rz 0.18 deg; joints [-7.835, -138.835, -56.669, -67.538, 92.098, -13.072]
  MoveL 2016 to (170.19, -150.75, 369) mm, rotated rx -22.61 ry -0.43 rz 0.18 deg; joints [-7.591, -137.767, -58.693, -66.425, 92.092, -12.826]
  MoveL 2017 to (175.97, -149.23, 370) mm, rotated rx -22.69 ry -0.32 rz 0.13 deg; joints [-7.964, -138.057, -58.383, -66.511, 92.005, -13.198]
  MoveL 2018 to (174.99, -144.5, 367.51) mm, rotated rx -22.62 ry -0.29 rz 0.12 deg; joints [-7.978, -137.206, -60.004, -65.666, 91.991, -13.21]
  MoveL 2019 to (174.96, -134.73, 361.78) mm, rotated rx -22.16 ry -0.69 rz 0.28 deg; joints [-8.379, -135.494, -63.25, -63.797, 92.57, -13.598]
  MoveL 2020 to (174.54, -127.59, 360.29) mm, rotated rx -22.11 ry -1.08 rz 0.44 deg; joints [-8.639, -134.746, -64.955, -62.902, 93.024, -13.86]
  MoveL 2021 to (175.78, -123.76, 358.52) mm, rotated rx -21.77 ry -1.43 rz 0.57 deg; joints [-8.987, -134.2, -66.103, -62.081, 93.52, -14.2]
  MoveL 2022 to (175.03, -115.54, 355.67) mm, rotated rx -21.4 ry -2.19 rz 0.86 deg; joints [-9.448, -133.171, -68.317, -60.755, 94.459, -14.659]
  MoveL 2023 to (175.49, -107.34, 350.83) mm, rotated rx -21.09 ry -2.91 rz 1.12 deg; joints [-10.007, -132.056, -70.388, -59.733, 95.357, -15.22]
  MoveL 2024 to (174.49, -102.27, 348.62) mm, rotated rx -21.14 ry -3.01 rz 1.16 deg; joints [-10.083, -131.424, -71.586, -59.258, 95.457, -15.3]
  MoveL 2025 to (175.17, -94.45, 346.42) mm, rotated rx -21 ry -3.25 rz 1.25 deg; joints [-10.417, -130.627, -73.363, -58.234, 95.786, -15.634]
  MoveL 2026 to (175.06, -84.76, 343.57) mm, rotated rx -20.58 ry -3.18 rz 1.19 deg; joints [-10.637, -129.406, -76.061, -56.355, 95.856, -15.836]
  MoveL 2027 to (175.57, -77.85, 340.28) mm, rotated rx -20.47 ry -3.22 rz 1.2 deg; joints [-10.874, -128.555, -77.691, -55.502, 95.954, -16.068]
  MoveL 2028 to (174.52, -73.06, 337.84) mm, rotated rx -20.59 ry -3.02 rz 1.13 deg; joints [-10.812, -127.907, -78.828, -55.07, 95.706, -16.005]
  MoveL 2029 to (174.82, -64.84, 334.43) mm, rotated rx -21.45 ry -2.71 rz 1.07 deg; joints [-10.806, -127.277, -79.786, -55.486, 95.173, -16.023]
  MoveL 2030 to (175.03, -55.06, 332.28) mm, rotated rx -20.34 ry -2.65 rz 0.98 deg; joints [-11.141, -125.966, -82.992, -52.532, 95.44, -16.311]
  MoveL 2031 to (174.79, -47.9, 330.15) mm, rotated rx -19.13 ry -2.62 rz 0.91 deg; joints [-11.426, -124.836, -85.733, -49.769, 95.776, -16.538]
  MoveL 2032 to (175.14, -43.31, 326.9) mm, rotated rx -18.54 ry -2.58 rz 0.87 deg; joints [-11.649, -124.013, -87.309, -48.457, 95.936, -16.727]
  MoveL 2033 to (175.22, -34.93, 324.04) mm, rotated rx -18.61 ry -2.4 rz 0.81 deg; joints [-11.781, -123.207, -88.95, -47.646, 95.752, -16.856]
  MoveL 2034 to (175.12, -24.65, 322.03) mm, rotated rx -19.11 ry -2.21 rz 0.76 deg; joints [-11.877, -122.538, -90.456, -47.246, 95.439, -16.971]
  MoveL 2035 to (177.03, -17.59, 320.12) mm, rotated rx -18.53 ry -2.16 rz 0.72 deg; joints [-12.278, -121.861, -92.181, -45.665, 95.621, -17.337]
  MoveL 2036 to (174.49, -13.29, 317.96) mm, rotated rx -18.44 ry -1.83 rz 0.61 deg; joints [-12.048, -121.162, -93.472, -44.867, 95.277, -17.094]
  MoveL 2037 to (175.18, -4.27, 314.07) mm, rotated rx -19.38 ry -1.35 rz 0.48 deg; joints [-12.011, -120.467, -94.437, -45.357, 94.518, -17.096]
  MoveL 2038 to (174.91, 5.34, 311.34) mm, rotated rx -19.59 ry -1.35 rz 0.48 deg; joints [-12.222, -119.735, -95.999, -44.738, 94.488, -17.314]
  MoveL 2039 to (175.01, 15.24, 307.77) mm, rotated rx -19.46 ry -1.65 rz 0.58 deg; joints [-12.691, -118.904, -97.737, -43.844, 94.905, -17.78]
  MoveL 2040 to (175.09, 25.14, 304.17) mm, rotated rx -18.4 ry -1.93 rz 0.64 deg; joints [-13.31, -117.84, -100.294, -41.48, 95.618, -18.342]
  MoveL 2041 to (175.17, 33.6, 300.92) mm, rotated rx -17.79 ry -2.07 rz 0.66 deg; joints [-13.76, -116.993, -102.227, -39.897, 96.024, -18.755]
  MoveL 2042 to (175.02, 38.04, 299) mm, rotated rx -17.51 ry -2.09 rz 0.66 deg; joints [-13.957, -116.522, -103.231, -39.13, 96.169, -18.932]
  MoveL 2043 to (175, 44.8, 297.93) mm, rotated rx -17.36 ry -2.07 rz 0.65 deg; joints [-14.181, -116.102, -104.457, -38.196, 96.245, -19.143]
  MoveL 2044 to (174.86, 55.26, 294.85) mm, rotated rx -17.73 ry -1.98 rz 0.63 deg; joints [-14.41, -115.394, -105.909, -37.795, 96.073, -19.389]
  MoveL 2045 to (175.12, 64.56, 291.22) mm, rotated rx -18.61 ry -2.06 rz 0.69 deg; joints [-14.668, -114.84, -106.634, -38.518, 95.921, -19.702]
  MoveL 2046 to (174.84, 69.25, 289) mm, rotated rx -19.07 ry -2.11 rz 0.73 deg; joints [-14.767, -114.499, -107.028, -38.931, 95.837, -19.829]
  MoveL 2047 to (174.75, 74.88, 287.44) mm, rotated rx -19.13 ry -1.76 rz 0.61 deg; joints [-14.755, -114.031, -108.055, -38.304, 95.461, -19.809]
  MoveL 2048 to (175.06, 84.56, 284.73) mm, rotated rx -18.42 ry -1.65 rz 0.55 deg; joints [-15.21, -113.226, -110.191, -36.306, 95.672, -20.213]
  MoveL 2049 to (174.94, 94.08, 281.49) mm, rotated rx -18.01 ry -1.83 rz 0.6 deg; joints [-15.749, -112.493, -111.931, -35.033, 96.088, -20.725]
  MoveL 2050 to (173.89, 98.94, 279) mm, rotated rx -17.91 ry -1.78 rz 0.57 deg; joints [-15.843, -111.94, -112.917, -34.489, 96.084, -20.809]
  MoveL 2051 to (175.02, 104.79, 277.28) mm, rotated rx -17.74 ry -1.73 rz 0.55 deg; joints [-16.198, -111.582, -113.857, -33.769, 96.159, -21.146]
  MoveL 2052 to (174.82, 115.07, 274.4) mm, rotated rx -17.36 ry -1.56 rz 0.49 deg; joints [-16.585, -110.839, -115.791, -32.199, 96.206, -21.494]
  MoveL 2053 to (174.95, 124.61, 271.66) mm, rotated rx -16.79 ry -1.72 rz 0.52 deg; joints [-17.227, -110.238, -117.529, -30.664, 96.697, -22.092]
  MoveL 2054 to (174.52, 131.84, 271.21) mm, rotated rx -15.92 ry -1.63 rz 0.46 deg; joints [-17.607, -109.913, -119.269, -28.44, 97.003, -22.392]
  MoveL 2055 to (169.38, 132.93, 271) mm, rotated rx -15.41 ry -1.32 rz 0.36 deg; joints [-17.034, -109.463, -120.428, -27.074, 96.771, -21.771]
  MoveL 2056 to (184.4, -264.1, 413.76) mm, rotated rx -18.8 ry -1.23 rz 0.42 deg; joints [-7.311, -162.374, -9.621, -87.337, 93.702, -12.429]
  MoveL 2057 to (184.76, -255.49, 411.71) mm, rotated rx -20.31 ry -1.25 rz 0.46 deg; joints [-7.355, -161.876, -10.445, -88.497, 93.417, -12.529]
  MoveL 2058 to (184.38, -243.64, 408.04) mm, rotated rx -21.62 ry -2.19 rz 0.87 deg; joints [-7.749, -159.675, -14.822, -87.835, 94.185, -12.978]
  MoveL 2059 to (185.03, -234.87, 404.22) mm, rotated rx -22.26 ry -2.81 rz 1.15 deg; joints [-8.112, -157.612, -18.897, -86.625, 94.754, -13.369]
  MoveL 2060 to (178.74, -228.23, 400) mm, rotated rx -21.99 ry -2.76 rz 1.11 deg; joints [-7.828, -153.767, -26.585, -82.483, 94.718, -13.078]
  MoveL 2061 to (185.81, -227.58, 400.43) mm, rotated rx -21.9 ry -2.95 rz 1.18 deg; joints [-8.363, -154.403, -25.451, -82.976, 95, -13.611]
  MoveL 2062 to (184.34, -222.82, 398.55) mm, rotated rx -21.59 ry -2.84 rz 1.12 deg; joints [-8.33, -152.38, -29.651, -80.471, 94.945, -13.566]
  MoveL 2063 to (185.03, -214.73, 396.61) mm, rotated rx -21.31 ry -2.69 rz 1.05 deg; joints [-8.467, -150.17, -34.406, -77.629, 94.868, -13.691]
  MoveL 2064 to (184.94, -204.58, 392.87) mm, rotated rx -22.13 ry -1.58 rz 0.64 deg; joints [-8.153, -148.278, -38.083, -76.356, 93.488, -13.385]
  MoveL 2065 to (183.95, -198.06, 390) mm, rotated rx -23.1 ry -0.72 rz 0.31 deg; joints [-7.794, -147.382, -39.633, -76.431, 92.32, -13.044]
  MoveL 2066 to (185.57, -194.26, 387.77) mm, rotated rx -23.43 ry -0.39 rz 0.17 deg; joints [-7.819, -146.81, -40.635, -76.239, 91.904, -13.074]
  MoveL 2067 to (184.84, -185.7, 383.39) mm, rotated rx -23.22 ry -0.59 rz 0.25 deg; joints [-8.014, -144.877, -44.445, -74.217, 92.18, -13.264]
  MoveL 2068 to (183.16, -178.67, 380.27) mm, rotated rx -22.68 ry -0.83 rz 0.35 deg; joints [-8.161, -143.12, -48.056, -71.898, 92.57, -13.399]
  MoveL 2069 to (185.13, -173.59, 378.32) mm, rotated rx -22.21 ry -1.16 rz 0.47 deg; joints [-8.555, -142.151, -50.146, -70.414, 93.074, -13.78]
  MoveL 2070 to (185.24, -164.63, 375.93) mm, rotated rx -22.18 ry -1.22 rz 0.5 deg; joints [-8.745, -140.845, -52.953, -68.913, 93.175, -13.969]
  MoveL 2071 to (185.14, -154.81, 371.89) mm, rotated rx -22.82 ry -1.22 rz 0.51 deg; joints [-8.865, -139.74, -54.999, -68.61, 93.039, -14.107]
  MoveL 2072 to (181.77, -149.23, 370) mm, rotated rx -22.81 ry -0.85 rz 0.36 deg; joints [-8.58, -138.619, -57.271, -67.337, 92.613, -13.819]
  MoveL 2073 to (185.43, -144.58, 366.07) mm, rotated rx -22.78 ry -1.22 rz 0.51 deg; joints [-9.098, -138.017, -58.204, -67.095, 93.07, -14.337]
  MoveL 2074 to (184.98, -134.54, 360.83) mm, rotated rx -21.81 ry -1 rz 0.4 deg; joints [-9.278, -135.81, -62.661, -63.854, 93.101, -14.483]
  MoveL 2075 to (184.16, -124.99, 358.51) mm, rotated rx -21.12 ry -1.67 rz 0.65 deg; joints [-9.742, -134.479, -65.719, -61.664, 94.028, -14.93]
  MoveL 2076 to (184.81, -115.61, 355.69) mm, rotated rx -20.32 ry -2.95 rz 1.09 deg; joints [-10.593, -133.382, -68.299, -59.814, 95.671, -15.774]
  MoveL 2077 to (185.46, -104.79, 350.86) mm, rotated rx -20.81 ry -3.77 rz 1.43 deg; joints [-11.187, -132.515, -69.834, -59.918, 96.481, -16.411]
  MoveL 2078 to (180.81, -101.08, 349) mm, rotated rx -20.89 ry -3.49 rz 1.33 deg; joints [-10.804, -131.726, -71.266, -59.233, 96.115, -16.022]
  MoveL 2079 to (184.68, -94.44, 347.4) mm, rotated rx -20.81 ry -3.92 rz 1.49 deg; joints [-11.429, -131.346, -72.262, -58.724, 96.665, -16.657]
  MoveL 2080 to (184.77, -84.65, 343.4) mm, rotated rx -20.87 ry -3.6 rz 1.37 deg; joints [-11.532, -130.139, -74.607, -57.571, 96.334, -16.751]
  MoveL 2081 to (185.52, -76.52, 340.59) mm, rotated rx -21.14 ry -2.9 rz 1.12 deg; joints [-11.449, -129.219, -76.407, -56.735, 95.527, -16.657]
  MoveL 2082 to (184.05, -71.92, 338.65) mm, rotated rx -21.36 ry -2.65 rz 1.04 deg; joints [-11.317, -128.639, -77.452, -56.399, 95.196, -16.528]
  MoveL 2083 to (184.99, -65.35, 335.87) mm, rotated rx -21.41 ry -2.34 rz 0.92 deg; joints [-11.411, -127.879, -78.912, -55.665, 94.871, -16.615]
  MoveL 2084 to (184.93, -55.01, 332.63) mm, rotated rx -20.15 ry -2.74 rz 1 deg; joints [-11.99, -126.464, -82.234, -52.717, 95.71, -17.149]
  MoveL 2085 to (184.59, -43.77, 327.5) mm, rotated rx -18.81 ry -2.78 rz 0.95 deg; joints [-12.461, -124.736, -85.97, -49.479, 96.203, -17.552]
  MoveL 2086 to (185.18, -34.99, 325.03) mm, rotated rx -18.69 ry -2.53 rz 0.85 deg; joints [-12.641, -123.894, -87.855, -48.26, 96.012, -17.716]
  MoveL 2087 to (185.09, -24.65, 322.18) mm, rotated rx -19.12 ry -2.6 rz 0.9 deg; joints [-12.89, -123.173, -89.348, -47.955, 96, -17.988]
